LIN {X 4.349,Y -47.961,Z -134.902,A -90.000,B 90.000,C 0.000} C_DIS
LIN {X 3.638,Y -47.921,Z -134.978,A -90.000,B 90.000,C 0.000} C_DIS
LIN {X 3.458,Y -47.911,Z -134.966,A -90.000,B 90.000,C 0.000} C_DIS
LIN {X 3.249,Y -47.899,Z -134.959,A -90.000,B 90.000,C 0.000} C_DIS
LIN {X 3.035,Y -47.886,Z -134.959,A -90.000,B 90.000,C 0.000} C_DIS
LIN {X 2.734,Y -47.862,Z -134.966,A -90.000,B 90.000,C 0.000} C_DIS
LIN {X 2.521,Y -47.844,Z -134.907,A -90.000,B 90.000,C 0.000} C_DIS
LIN {X 2.240,Y -47.821,Z -134.818,A -90.000,B 90.000,C 0.000} C_DIS
LIN {X 1.961,Y -47.797,Z -134.712,A -90.000,B 90.000,C 0.000} C_DIS
LIN {X 1.753,Y -47.779,Z -134.622,A -90.000,B 90.000,C 0.000} C_DIS
LIN {X 1.325,Y -47.740,Z -134.399,A -90.000,B 90.000,C 0.000} C_DIS
LIN {X 1.040,Y -47.714,Z -134.237,A -90.000,B 90.000,C 0.000} C_DIS
LIN {X 0.850,Y -47.696,Z -134.116,A -90.000,B 90.000,C 0.000} C_DIS
LIN {X 0.755,Y -47.686,Z -134.050,A -90.000,B 90.000,C 0.000} C_DIS
LIN {X 0.661,Y -47.677,Z -133.981,A -90.000,B 90.000,C 0.000} C_DIS
LIN {X 0.569,Y -47.666,Z -133.907,A -90.000,B 90.000,C 0.000} C_DIS
LIN {X 0.394,Y -47.651,Z -133.762,A -90.000,B 90.000,C 0.000} C_DIS
LIN {X 0.029,Y -47.630,Z -133.079,A -90.000,B 90.000,C 0.000} C_DIS
LIN {X -0.030,Y -47.623,Z -132.969,A -90.000,B 90.000,C 0.000} C_DIS
LIN {X -0.099,Y -47.611,Z -132.836,A -90.000,B 90.000,C 0.000} C_DIS
LIN {X -0.133,Y -47.605,Z -132.740,A -90.000,B 90.000,C 0.000} C_DIS
LIN {X 0.043,Y -47.607,Z -130.577,A -90.000,B 90.000,C 0.000} C_DIS
LIN {X 0.099,Y -47.612,Z -130.301,A -90.000,B 90.000,C 0.000} C_DIS
LIN {X 0.135,Y -47.611,Z -130.125,A -90.000,B 90.000,C 0.000} C_DIS
LIN {X 0.250,Y -47.612,Z -129.925,A -90.000,B 90.000,C 0.000} C_DIS
LIN {X 1.143,Y -47.614,Z -128.527,A -90.000,B 90.000,C 0.000} C_DIS
LIN {X 1.838,Y -47.607,Z -127.443,A -90.000,B 90.000,C 0.000} C_DIS
LIN {X 2.056,Y -47.610,Z -127.175,A -90.000,B 90.000,C 0.000} C_DIS
LIN {X 2.200,Y -47.615,Z -127.035,A -90.000,B 90.000,C 0.000} C_DIS
LIN {X 2.268,Y -47.616,Z -126.970,A -90.000,B 90.000,C 0.000} C_DIS
LIN {X 3.440,Y -47.612,Z -125.853,A -90.000,B 90.000,C 0.000} C_DIS
LIN {X 3.637,Y -47.607,Z -125.667,A -90.000,B 90.000,C 0.000} C_DIS
LIN {X 4.260,Y -47.595,Z -125.097,A -90.000,B 90.000,C 0.000} C_DIS
LIN {X 4.386,Y -47.595,Z -125.003,A -90.000,B 90.000,C 0.000} C_DIS
LIN {X 5.546,Y -47.602,Z -124.204,A -90.000,B 90.000,C 0.000} C_DIS
LIN {X 5.853,Y -47.602,Z -123.993,A -90.000,B 90.000,C 0.000} C_DIS
LIN {X 6.516,Y -47.588,Z -123.540,A -90.000,B 90.000,C 0.000} C_DIS
LIN {X 6.563,Y -47.588,Z -123.512,A -90.000,B 90.000,C 0.000} C_DIS
LIN {X 8.622,Y -47.571,Z -122.476,A -90.000,B 90.000,C 0.000} C_DIS
LIN {X 9.750,Y -47.547,Z -121.910,A -90.000,B 90.000,C 0.000} C_DIS
LIN {X 12.160,Y -47.550,Z -121.167,A -90.000,B 90.000,C 0.000} C_DIS
LIN {X 14.408,Y -47.502,Z -120.480,A -90.000,B 90.000,C 0.000} C_DIS
LIN {X 14.547,Y -47.502,Z -120.468,A -90.000,B 90.000,C 0.000} C_DIS
LIN {X 16.833,Y -47.499,Z -120.228,A -90.000,B 90.000,C 0.000} C_DIS
LIN {X 17.033,Y -47.496,Z -120.208,A -90.000,B 90.000,C 0.000} C_DIS
LIN {X 18.502,Y -47.463,Z -120.057,A -90.000,B 90.000,C 0.000} C_DIS
LIN {X 18.616,Y -47.461,Z -120.057,A -90.000,B 90.000,C 0.000} C_DIS
LIN {X 21.308,Y -47.456,Z -120.534,A -90.000,B 90.000,C 0.000} C_DIS
LIN {X 21.567,Y -47.448,Z -120.581,A -90.000,B 90.000,C 0.000} C_DIS
LIN {X 21.787,Y -47.441,Z -120.626,A -90.000,B 90.000,C 0.000} C_DIS
LIN {X 22.175,Y -47.441,Z -120.928,A -90.000,B 90.000,C 0.000} C_DIS
LIN {X 23.178,Y -47.428,Z -121.711,A -90.000,B 90.000,C 0.000} C_DIS
LIN {X 23.442,Y -47.428,Z -122.009,A -90.000,B 90.000,C 0.000} C_DIS
LIN {X 23.523,Y -47.442,Z -122.462,A -90.000,B 90.000,C 0.000} C_DIS
LIN {X 23.482,Y -47.463,Z -122.835,A -90.000,B 90.000,C 0.000} C_DIS
LIN {X 23.458,Y -47.474,Z -123.058,A -90.000,B 90.000,C 0.000} C_DIS
LIN {X 23.449,Y -47.486,Z -123.390,A -90.000,B 90.000,C 0.000} C_DIS
LIN {X 23.488,Y -47.490,Z -123.844,A -90.000,B 90.000,C 0.000} C_DIS
LIN {X 23.560,Y -47.491,Z -124.679,A -90.000,B 90.000,C 0.000} C_DIS
LIN {X 23.397,Y -47.512,Z -125.426,A -90.000,B 90.000,C 0.000} C_DIS
LIN {X 23.214,Y -47.513,Z -126.253,A -90.000,B 90.000,C 0.000} C_DIS
LIN {X 23.157,Y -47.516,Z -126.512,A -90.000,B 90.000,C 0.000} C_DIS
LIN {X 22.471,Y -47.582,Z -127.926,A -90.000,B 90.000,C 0.000} C_DIS
LIN {X 22.078,Y -47.598,Z -128.731,A -90.000,B 90.000,C 0.000} C_DIS
LIN {X 21.868,Y -47.607,Z -129.140,A -90.000,B 90.000,C 0.000} C_DIS
LIN {X 21.688,Y -47.619,Z -129.394,A -90.000,B 90.000,C 0.000} C_DIS
LIN {X 20.899,Y -47.663,Z -130.579,A -90.000,B 90.000,C 0.000} C_DIS
LIN {X 20.391,Y -47.672,Z -131.337,A -90.000,B 90.000,C 0.000} C_DIS
LIN {X 19.805,Y -47.696,Z -132.023,A -90.000,B 90.000,C 0.000} C_DIS
LIN {X 19.346,Y -47.720,Z -132.478,A -90.000,B 90.000,C 0.000} C_DIS
LIN {X 18.457,Y -47.730,Z -133.348,A -90.000,B 90.000,C 0.000} C_DIS
LIN {X 18.205,Y -47.729,Z -133.593,A -90.000,B 90.000,C 0.000} C_DIS
LIN {X 17.590,Y -47.732,Z -134.145,A -90.000,B 90.000,C 0.000} C_DIS
LIN {X 17.544,Y -47.732,Z -134.183,A -90.000,B 90.000,C 0.000} C_DIS
LIN {X 17.409,Y -47.738,Z -134.263,A -90.000,B 90.000,C 0.000} C_DIS
LIN {X 17.214,Y -47.749,Z -134.364,A -90.000,B 90.000,C 0.000} C_DIS
LIN {X 16.932,Y -47.764,Z -134.516,A -90.000,B 90.000,C 0.000} C_DIS
LIN {X 16.164,Y -47.806,Z -134.922,A -90.000,B 90.000,C 0.000} C_DIS
LIN {X 15.908,Y -47.817,Z -135.056,A -90.000,B 90.000,C 0.000} C_DIS
LIN {X 15.083,Y -47.818,Z -135.479,A -90.000,B 90.000,C 0.000} C_DIS
LIN {X 14.959,Y -47.815,Z -135.542,A -90.000,B 90.000,C 0.000} C_DIS
LIN {X 13.972,Y -47.784,Z -136.033,A -90.000,B 90.000,C 0.000} C_DIS
LIN {X 13.915,Y -47.784,Z -136.053,A -90.000,B 90.000,C 0.000} C_DIS
LIN {X 13.450,Y -47.784,Z -136.207,A -90.000,B 90.000,C 0.000} C_DIS
LIN {X 13.362,Y -47.784,Z -136.234,A -90.000,B 90.000,C 0.000} C_DIS
LIN {X 13.341,Y -47.785,Z -136.240,A -90.000,B 90.000,C 0.000} C_DIS
LIN {X 12.439,Y -47.811,Z -136.397,A -90.000,B 90.000,C 0.000} C_DIS
LIN {X 10.398,Y -47.880,Z -136.688,A -90.000,B 90.000,C 0.000} C_DIS
LIN {X 10.207,Y -47.881,Z -136.713,A -90.000,B 90.000,C 0.000} C_DIS
LIN {X 9.590,Y -47.863,Z -136.790,A -90.000,B 90.000,C 0.000} C_DIS
LIN {X 8.229,Y -47.857,Z -136.774,A -90.000,B 90.000,C 0.000} C_DIS
LIN {X 7.049,Y -47.839,Z -136.755,A -90.000,B 90.000,C 0.000} C_DIS
LIN {X 6.522,Y -47.832,Z -136.740,A -90.000,B 90.000,C 0.000} C_DIS
LIN {X 6.298,Y -47.824,Z -136.732,A -90.000,B 90.000,C 0.000} C_DIS
LIN {X 6.019,Y -47.803,Z -136.719,A -90.000,B 90.000,C 0.000} C_DIS
LIN {X 5.735,Y -47.783,Z -136.693,A -90.000,B 90.000,C 0.000} C_DIS
LIN {X 5.512,Y -47.783,Z -136.604,A -90.000,B 90.000,C 0.000} C_DIS
LIN {X 5.374,Y -47.782,Z -136.555,A -90.000,B 90.000,C 0.000} C_DIS
LIN {X 3.264,Y -47.744,Z -135.889,A -90.000,B 90.000,C 0.000} C_DIS
LIN {X 3.000,Y -47.743,Z -135.807,A -90.000,B 90.000,C 0.000} C_DIS
LIN {X 2.785,Y -47.739,Z -135.739,A -90.000,B 90.000,C 0.000} C_DIS
LIN {X 2.660,Y -47.732,Z -135.698,A -90.000,B 90.000,C 0.000} C_DIS
LIN {X 2.579,Y -47.735,Z -135.627,A -90.000,B 90.000,C 0.000} C_DIS
LIN {X 2.188,Y -47.735,Z -135.280,A -90.000,B 90.000,C 0.000} C_DIS
LIN {X 1.658,Y -47.726,Z -134.806,A -90.000,B 90.000,C 0.000} C_DIS
LIN {X 1.300,Y -47.717,Z -134.512,A -90.000,B 90.000,C 0.000} C_DIS
LIN {X 1.078,Y -47.706,Z -134.329,A -90.000,B 90.000,C 0.000} C_DIS
LIN {X 0.956,Y -47.697,Z -134.228,A -90.000,B 90.000,C 0.000} C_DIS
LIN {X 0.569,Y -47.666,Z -133.907,A -90.000,B 90.000,C 0.000} C_DIS
LIN {X 0.393,Y -47.657,Z -133.765,A -90.000,B 90.000,C 0.000} C_DIS
LIN {X 0.270,Y -47.647,Z -133.556,A -90.000,B 90.000,C 0.000} C_DIS
LIN {X 0.189,Y -47.641,Z -133.425,A -90.000,B 90.000,C 0.000} C_DIS
LIN {X 0.021,Y -47.629,Z -133.169,A -90.000,B 90.000,C 0.000} C_DIS
LIN {X -0.161,Y -47.616,Z -132.904,A -90.000,B 90.000,C 0.000} C_DIS
LIN {X -0.203,Y -47.612,Z -132.822,A -90.000,B 90.000,C 0.000} C_DIS
LIN {X -0.214,Y -47.605,Z -132.651,A -90.000,B 90.000,C 0.000} C_DIS
LIN {X -0.228,Y -47.600,Z -132.517,A -90.000,B 90.000,C 0.000} C_DIS
LIN {X -0.255,Y -47.592,Z -132.319,A -90.000,B 90.000,C 0.000} C_DIS
LIN {X -0.278,Y -47.586,Z -132.189,A -90.000,B 90.000,C 0.000} C_DIS
LIN {X -0.318,Y -47.579,Z -131.998,A -90.000,B 90.000,C 0.000} C_DIS
LIN {X -0.349,Y -47.573,Z -131.872,A -90.000,B 90.000,C 0.000} C_DIS
LIN {X -0.420,Y -47.563,Z -131.624,A -90.000,B 90.000,C 0.000} C_DIS
LIN {X -0.560,Y -47.540,Z -131.077,A -90.000,B 90.000,C 0.000} C_DIS
LIN {X -0.623,Y -47.526,Z -130.741,A -90.000,B 90.000,C 0.000} C_DIS
LIN {X -0.614,Y -47.515,Z -130.467,A -90.000,B 90.000,C 0.000} C_DIS
LIN {X -0.615,Y -47.511,Z -130.363,A -90.000,B 90.000,C 0.000} C_DIS
LIN {X -0.627,Y -47.502,Z -130.152,A -90.000,B 90.000,C 0.000} C_DIS
LIN {X -0.654,Y -47.493,Z -129.936,A -90.000,B 90.000,C 0.000} C_DIS
LIN {X -0.672,Y -47.488,Z -129.827,A -90.000,B 90.000,C 0.000} C_DIS
LIN {X -0.704,Y -47.480,Z -129.660,A -90.000,B 90.000,C 0.000} C_DIS
LIN {X -0.743,Y -47.466,Z -129.380,A -90.000,B 90.000,C 0.000} C_DIS
LIN {X -0.791,Y -47.452,Z -129.092,A -90.000,B 90.000,C 0.000} C_DIS
LIN {X -0.801,Y -47.447,Z -128.991,A -90.000,B 90.000,C 0.000} C_DIS
LIN {X -0.783,Y -47.438,Z -128.816,A -90.000,B 90.000,C 0.000} C_DIS
LIN {X -0.768,Y -47.433,Z -128.708,A -90.000,B 90.000,C 0.000} C_DIS
LIN {X -0.752,Y -47.427,Z -128.600,A -90.000,B 90.000,C 0.000} C_DIS
LIN {X -0.728,Y -47.422,Z -128.495,A -90.000,B 90.000,C 0.000} C_DIS
LIN {X -0.671,Y -47.411,Z -128.283,A -90.000,B 90.000,C 0.000} C_DIS
LIN {X -0.604,Y -47.400,Z -128.068,A -90.000,B 90.000,C 0.000} C_DIS
LIN {X -0.529,Y -47.389,Z -127.846,A -90.000,B 90.000,C 0.000} C_DIS
LIN {X -0.445,Y -47.377,Z -127.616,A -90.000,B 90.000,C 0.000} C_DIS
LIN {X -0.351,Y -47.364,Z -127.380,A -90.000,B 90.000,C 0.000} C_DIS
LIN {X -0.299,Y -47.358,Z -127.259,A -90.000,B 90.000,C 0.000} C_DIS
LIN {X -0.184,Y -47.345,Z -127.012,A -90.000,B 90.000,C 0.000} C_DIS
LIN {X -0.053,Y -47.331,Z -126.758,A -90.000,B 90.000,C 0.000} C_DIS
LIN {X 0.020,Y -47.323,Z -126.629,A -90.000,B 90.000,C 0.000} C_DIS
LIN {X 0.179,Y -47.308,Z -126.366,A -90.000,B 90.000,C 0.000} C_DIS
LIN {X 0.233,Y -47.308,Z -126.282,A -90.000,B 90.000,C 0.000} C_DIS
LIN {X 0.581,Y -47.308,Z -125.855,A -90.000,B 90.000,C 0.000} C_DIS
LIN {X 0.688,Y -47.308,Z -125.746,A -90.000,B 90.000,C 0.000} C_DIS
LIN {X 2.304,Y -47.308,Z -124.205,A -90.000,B 90.000,C 0.000} C_DIS
LIN {X 2.998,Y -47.308,Z -123.569,A -90.000,B 90.000,C 0.000} C_DIS
LIN {X 3.235,Y -47.308,Z -123.392,A -90.000,B 90.000,C 0.000} C_DIS
LIN {X 5.471,Y -47.308,Z -121.855,A -90.000,B 90.000,C 0.000} C_DIS
LIN {X 5.627,Y -47.308,Z -121.766,A -90.000,B 90.000,C 0.000} C_DIS
LIN {X 9.005,Y -47.308,Z -120.061,A -90.000,B 90.000,C 0.000} C_DIS
LIN {X 13.904,Y -47.308,Z -118.552,A -90.000,B 90.000,C 0.000} C_DIS
LIN {X 14.072,Y -47.308,Z -118.512,A -90.000,B 90.000,C 0.000} C_DIS
LIN {X 14.371,Y -47.308,Z -118.485,A -90.000,B 90.000,C 0.000} C_DIS
LIN {X 18.398,Y -47.308,Z -118.063,A -90.000,B 90.000,C 0.000} C_DIS
LIN {X 18.792,Y -47.308,Z -118.063,A -90.000,B 90.000,C 0.000} C_DIS
LIN {X 21.939,Y -47.308,Z -118.620,A -90.000,B 90.000,C 0.000} C_DIS
LIN {X 22.643,Y -47.308,Z -118.763,A -90.000,B 90.000,C 0.000} C_DIS
LIN {X 24.510,Y -47.308,Z -120.218,A -90.000,B 90.000,C 0.000} C_DIS
LIN {X 24.576,Y -47.308,Z -120.277,A -90.000,B 90.000,C 0.000} C_DIS
LIN {X 25.298,Y -47.308,Z -121.096,A -90.000,B 90.000,C 0.000} C_DIS
LIN {X 25.323,Y -47.308,Z -121.181,A -90.000,B 90.000,C 0.000} C_DIS
LIN {X 25.538,Y -47.308,Z -122.399,A -90.000,B 90.000,C 0.000} C_DIS
LIN {X 25.438,Y -47.308,Z -123.282,A -90.000,B 90.000,C 0.000} C_DIS
LIN {X 25.566,Y -47.308,Z -124.764,A -90.000,B 90.000,C 0.000} C_DIS
LIN {X 25.558,Y -47.308,Z -124.867,A -90.000,B 90.000,C 0.000} C_DIS
LIN {X 25.073,Y -47.308,Z -127.058,A -90.000,B 90.000,C 0.000} C_DIS
LIN {X 25.021,Y -47.308,Z -127.227,A -90.000,B 90.000,C 0.000} C_DIS
LIN {X 25.004,Y -47.308,Z -127.267,A -90.000,B 90.000,C 0.000} C_DIS
LIN {X 24.995,Y -47.308,Z -127.282,A -90.000,B 90.000,C 0.000} C_DIS
LIN {X 23.838,Y -47.308,Z -129.636,A -90.000,B 90.000,C 0.000} C_DIS
LIN {X 23.694,Y -47.308,Z -129.917,A -90.000,B 90.000,C 0.000} C_DIS
LIN {X 23.558,Y -47.308,Z -130.176,A -90.000,B 90.000,C 0.000} C_DIS
LIN {X 23.296,Y -47.308,Z -130.542,A -90.000,B 90.000,C 0.000} C_DIS
LIN {X 21.965,Y -47.308,Z -132.519,A -90.000,B 90.000,C 0.000} C_DIS
LIN {X 21.855,Y -47.308,Z -132.651,A -90.000,B 90.000,C 0.000} C_DIS
LIN {X 21.236,Y -47.308,Z -133.369,A -90.000,B 90.000,C 0.000} C_DIS
LIN {X 19.541,Y -47.308,Z -135.022,A -90.000,B 90.000,C 0.000} C_DIS
LIN {X 18.869,Y -47.308,Z -135.624,A -90.000,B 90.000,C 0.000} C_DIS
LIN {X 18.653,Y -47.308,Z -135.802,A -90.000,B 90.000,C 0.000} C_DIS
LIN {X 18.421,Y -47.308,Z -135.934,A -90.000,B 90.000,C 0.000} C_DIS
LIN {X 17.821,Y -47.308,Z -136.249,A -90.000,B 90.000,C 0.000} C_DIS
LIN {X 15.640,Y -47.308,Z -137.367,A -90.000,B 90.000,C 0.000} C_DIS
LIN {X 14.735,Y -47.308,Z -137.824,A -90.000,B 90.000,C 0.000} C_DIS
LIN {X 14.524,Y -47.308,Z -137.898,A -90.000,B 90.000,C 0.000} C_DIS
LIN {X 13.952,Y -47.308,Z -138.087,A -90.000,B 90.000,C 0.000} C_DIS
LIN {X 13.796,Y -47.308,Z -138.129,A -90.000,B 90.000,C 0.000} C_DIS
LIN {X 13.757,Y -47.308,Z -138.140,A -90.000,B 90.000,C 0.000} C_DIS
LIN {X 12.690,Y -47.308,Z -138.317,A -90.000,B 90.000,C 0.000} C_DIS
LIN {X 9.707,Y -47.308,Z -138.712,A -90.000,B 90.000,C 0.000} C_DIS
LIN {X 7.282,Y -47.308,Z -138.687,A -90.000,B 90.000,C 0.000} C_DIS
LIN {X 7.000,Y -47.308,Z -138.683,A -90.000,B 90.000,C 0.000} C_DIS
LIN {X 5.923,Y -47.308,Z -138.655,A -90.000,B 90.000,C 0.000} C_DIS
LIN {X 5.452,Y -47.308,Z -138.620,A -90.000,B 90.000,C 0.000} C_DIS
LIN {X 5.219,Y -47.308,Z -138.578,A -90.000,B 90.000,C 0.000} C_DIS
LIN {X 4.796,Y -47.308,Z -138.410,A -90.000,B 90.000,C 0.000} C_DIS
LIN {X 1.927,Y -47.308,Z -137.517,A -90.000,B 90.000,C 0.000} C_DIS
LIN {X 1.708,Y -47.308,Z -137.427,A -90.000,B 90.000,C 0.000} C_DIS
LIN {X 1.512,Y -47.308,Z -137.293,A -90.000,B 90.000,C 0.000} C_DIS
LIN {X 0.365,Y -47.308,Z -136.273,A -90.000,B 90.000,C 0.000} C_DIS
LIN {X -1.002,Y -47.308,Z -135.167,A -90.000,B 90.000,C 0.000} C_DIS
LIN {X -1.165,Y -47.308,Z -134.995,A -90.000,B 90.000,C 0.000} C_DIS
LIN {X -1.289,Y -47.308,Z -134.793,A -90.000,B 90.000,C 0.000} C_DIS
LIN {X -1.910,Y -47.308,Z -133.644,A -90.000,B 90.000,C 0.000} C_DIS
LIN {X -2.118,Y -47.308,Z -133.061,A -90.000,B 90.000,C 0.000} C_DIS
LIN {X -2.129,Y -47.308,Z -132.882,A -90.000,B 90.000,C 0.000} C_DIS
LIN {X -1.918,Y -47.308,Z -130.298,A -90.000,B 90.000,C 0.000} C_DIS
LIN {X -1.761,Y -47.308,Z -129.531,A -90.000,B 90.000,C 0.000} C_DIS
LIN {X -1.718,Y -47.308,Z -129.388,A -90.000,B 90.000,C 0.000} C_DIS
LIN {X -1.614,Y -47.308,Z -129.199,A -90.000,B 90.000,C 0.000} C_DIS
LIN {X -1.441,Y -47.308,Z -128.899,A -90.000,B 90.000,C 0.000} C_DIS
LIN {X 0.179,Y -47.308,Z -126.366,A -90.000,B 90.000,C 0.000} C_DIS
LIN {X 0.233,Y -47.313,Z -126.281,A -90.000,B 90.000,C 0.000} C_DIS
LIN {X 0.390,Y -47.313,Z -126.081,A -90.000,B 90.000,C 0.000} C_DIS
LIN {X 0.561,Y -47.310,Z -125.850,A -90.000,B 90.000,C 0.000} C_DIS
LIN {X 0.836,Y -47.303,Z -125.538,A -90.000,B 90.000,C 0.000} C_DIS
LIN {X 1.062,Y -47.297,Z -125.273,A -90.000,B 90.000,C 0.000} C_DIS
LIN {X 1.280,Y -47.290,Z -125.003,A -90.000,B 90.000,C 0.000} C_DIS
LIN {X 1.492,Y -47.281,Z -124.728,A -90.000,B 90.000,C 0.000} C_DIS
LIN {X 1.697,Y -47.271,Z -124.450,A -90.000,B 90.000,C 0.000} C_DIS
LIN {X 1.897,Y -47.262,Z -124.167,A -90.000,B 90.000,C 0.000} C_DIS
LIN {X 2.191,Y -47.248,Z -123.742,A -90.000,B 90.000,C 0.000} C_DIS
LIN {X 2.514,Y -47.232,Z -123.260,A -90.000,B 90.000,C 0.000} C_DIS
LIN {X 2.679,Y -47.224,Z -123.041,A -90.000,B 90.000,C 0.000} C_DIS
LIN {X 2.885,Y -47.215,Z -122.777,A -90.000,B 90.000,C 0.000} C_DIS
LIN {X 3.512,Y -47.187,Z -122.001,A -90.000,B 90.000,C 0.000} C_DIS
LIN {X 3.933,Y -47.169,Z -121.488,A -90.000,B 90.000,C 0.000} C_DIS
LIN {X 4.251,Y -47.156,Z -121.106,A -90.000,B 90.000,C 0.000} C_DIS
LIN {X 4.360,Y -47.151,Z -120.981,A -90.000,B 90.000,C 0.000} C_DIS
LIN {X 4.778,Y -47.134,Z -120.527,A -90.000,B 90.000,C 0.000} C_DIS
LIN {X 4.894,Y -47.129,Z -120.410,A -90.000,B 90.000,C 0.000} C_DIS
LIN {X 5.014,Y -47.125,Z -120.299,A -90.000,B 90.000,C 0.000} C_DIS
LIN {X 5.293,Y -47.115,Z -120.063,A -90.000,B 90.000,C 0.000} C_DIS
LIN {X 5.678,Y -47.101,Z -119.758,A -90.000,B 90.000,C 0.000} C_DIS
LIN {X 5.943,Y -47.092,Z -119.561,A -90.000,B 90.000,C 0.000} C_DIS
LIN {X 6.078,Y -47.088,Z -119.465,A -90.000,B 90.000,C 0.000} C_DIS
LIN {X 6.353,Y -47.079,Z -119.275,A -90.000,B 90.000,C 0.000} C_DIS
LIN {X 6.494,Y -47.074,Z -119.183,A -90.000,B 90.000,C 0.000} C_DIS
LIN {X 6.782,Y -47.065,Z -119.002,A -90.000,B 90.000,C 0.000} C_DIS
LIN {X 7.079,Y -47.055,Z -118.828,A -90.000,B 90.000,C 0.000} C_DIS
LIN {X 7.231,Y -47.050,Z -118.743,A -90.000,B 90.000,C 0.000} C_DIS
LIN {X 7.542,Y -47.041,Z -118.579,A -90.000,B 90.000,C 0.000} C_DIS
LIN {X 8.112,Y -47.042,Z -118.292,A -90.000,B 90.000,C 0.000} C_DIS
LIN {X 8.422,Y -47.046,Z -118.166,A -90.000,B 90.000,C 0.000} C_DIS
LIN {X 10.316,Y -47.086,Z -117.578,A -90.000,B 90.000,C 0.000} C_DIS
LIN {X 10.927,Y -47.095,Z -117.389,A -90.000,B 90.000,C 0.000} C_DIS
LIN {X 13.319,Y -47.092,Z -116.652,A -90.000,B 90.000,C 0.000} C_DIS
LIN {X 13.423,Y -47.092,Z -116.623,A -90.000,B 90.000,C 0.000} C_DIS
LIN {X 13.602,Y -47.094,Z -116.579,A -90.000,B 90.000,C 0.000} C_DIS
LIN {X 13.823,Y -47.096,Z -116.538,A -90.000,B 90.000,C 0.000} C_DIS
LIN {X 14.179,Y -47.104,Z -116.505,A -90.000,B 90.000,C 0.000} C_DIS
LIN {X 15.609,Y -47.133,Z -116.352,A -90.000,B 90.000,C 0.000} C_DIS
LIN {X 17.666,Y -47.130,Z -116.136,A -90.000,B 90.000,C 0.000} C_DIS
LIN {X 18.223,Y -47.133,Z -116.078,A -90.000,B 90.000,C 0.000} C_DIS
LIN {X 18.399,Y -47.134,Z -116.070,A -90.000,B 90.000,C 0.000} C_DIS
LIN {X 18.793,Y -47.139,Z -116.070,A -90.000,B 90.000,C 0.000} C_DIS
LIN {X 19.140,Y -47.146,Z -116.100,A -90.000,B 90.000,C 0.000} C_DIS
LIN {X 20.083,Y -47.169,Z -116.265,A -90.000,B 90.000,C 0.000} C_DIS
LIN {X 22.335,Y -47.177,Z -116.664,A -90.000,B 90.000,C 0.000} C_DIS
LIN {X 23.040,Y -47.180,Z -116.807,A -90.000,B 90.000,C 0.000} C_DIS
LIN {X 23.322,Y -47.183,Z -116.886,A -90.000,B 90.000,C 0.000} C_DIS
LIN {X 23.626,Y -47.189,Z -117.025,A -90.000,B 90.000,C 0.000} C_DIS
LIN {X 23.766,Y -47.193,Z -117.112,A -90.000,B 90.000,C 0.000} C_DIS
LIN {X 23.856,Y -47.195,Z -117.177,A -90.000,B 90.000,C 0.000} C_DIS
LIN {X 24.910,Y -47.194,Z -117.998,A -90.000,B 90.000,C 0.000} C_DIS
LIN {X 25.752,Y -47.189,Z -118.655,A -90.000,B 90.000,C 0.000} C_DIS
LIN {X 25.850,Y -47.188,Z -118.738,A -90.000,B 90.000,C 0.000} C_DIS
LIN {X 25.908,Y -47.188,Z -118.790,A -90.000,B 90.000,C 0.000} C_DIS
LIN {X 26.003,Y -47.188,Z -118.881,A -90.000,B 90.000,C 0.000} C_DIS
LIN {X 26.074,Y -47.189,Z -118.957,A -90.000,B 90.000,C 0.000} C_DIS
LIN {X 26.562,Y -47.192,Z -119.510,A -90.000,B 90.000,C 0.000} C_DIS
LIN {X 26.795,Y -47.179,Z -119.776,A -90.000,B 90.000,C 0.000} C_DIS
LIN {X 26.950,Y -47.168,Z -119.977,A -90.000,B 90.000,C 0.000} C_DIS
LIN {X 27.026,Y -47.162,Z -120.098,A -90.000,B 90.000,C 0.000} C_DIS
LIN {X 27.105,Y -47.158,Z -120.252,A -90.000,B 90.000,C 0.000} C_DIS
LIN {X 27.129,Y -47.157,Z -120.305,A -90.000,B 90.000,C 0.000} C_DIS
LIN {X 27.215,Y -47.154,Z -120.545,A -90.000,B 90.000,C 0.000} C_DIS
LIN {X 27.239,Y -47.153,Z -120.630,A -90.000,B 90.000,C 0.000} C_DIS
LIN {X 27.286,Y -47.152,Z -120.834,A -90.000,B 90.000,C 0.000} C_DIS
LIN {X 27.478,Y -47.151,Z -121.920,A -90.000,B 90.000,C 0.000} C_DIS
LIN {X 27.508,Y -47.147,Z -122.093,A -90.000,B 90.000,C 0.000} C_DIS
LIN {X 27.524,Y -47.144,Z -122.225,A -90.000,B 90.000,C 0.000} C_DIS
LIN {X 27.531,Y -47.142,Z -122.369,A -90.000,B 90.000,C 0.000} C_DIS
LIN {X 27.525,Y -47.141,Z -122.555,A -90.000,B 90.000,C 0.000} C_DIS
LIN {X 27.468,Y -47.141,Z -123.074,A -90.000,B 90.000,C 0.000} C_DIS
LIN {X 27.441,Y -47.141,Z -123.309,A -90.000,B 90.000,C 0.000} C_DIS
LIN {X 27.527,Y -47.123,Z -124.323,A -90.000,B 90.000,C 0.000} C_DIS
LIN {X 27.539,Y -47.114,Z -124.471,A -90.000,B 90.000,C 0.000} C_DIS
LIN {X 27.554,Y -47.099,Z -124.680,A -90.000,B 90.000,C 0.000} C_DIS
LIN {X 27.547,Y -47.084,Z -124.923,A -90.000,B 90.000,C 0.000} C_DIS
LIN {X 27.539,Y -47.079,Z -125.025,A -90.000,B 90.000,C 0.000} C_DIS
LIN {X 27.497,Y -47.068,Z -125.296,A -90.000,B 90.000,C 0.000} C_DIS
LIN {X 27.188,Y -47.028,Z -126.666,A -90.000,B 90.000,C 0.000} C_DIS
LIN {X 26.985,Y -46.969,Z -127.539,A -90.000,B 90.000,C 0.000} C_DIS
LIN {X 26.902,Y -46.953,Z -127.807,A -90.000,B 90.000,C 0.000} C_DIS
LIN {X 26.817,Y -46.943,Z -128.029,A -90.000,B 90.000,C 0.000} C_DIS
LIN {X 26.762,Y -46.939,Z -128.147,A -90.000,B 90.000,C 0.000} C_DIS
LIN {X 26.726,Y -46.939,Z -128.215,A -90.000,B 90.000,C 0.000} C_DIS
LIN {X 26.204,Y -46.937,Z -129.278,A -90.000,B 90.000,C 0.000} C_DIS
LIN {X 26.139,Y -46.936,Z -129.410,A -90.000,B 90.000,C 0.000} C_DIS
LIN {X 25.577,Y -46.892,Z -130.532,A -90.000,B 90.000,C 0.000} C_DIS
LIN {X 25.287,Y -46.873,Z -131.083,A -90.000,B 90.000,C 0.000} C_DIS
LIN {X 25.269,Y -46.872,Z -131.114,A -90.000,B 90.000,C 0.000} C_DIS
LIN {X 25.173,Y -46.870,Z -131.270,A -90.000,B 90.000,C 0.000} C_DIS
LIN {X 24.900,Y -46.871,Z -131.655,A -90.000,B 90.000,C 0.000} C_DIS
LIN {X 24.020,Y -46.825,Z -132.942,A -90.000,B 90.000,C 0.000} C_DIS
LIN {X 23.560,Y -46.796,Z -133.612,A -90.000,B 90.000,C 0.000} C_DIS
LIN {X 23.449,Y -46.793,Z -133.758,A -90.000,B 90.000,C 0.000} C_DIS
LIN {X 23.317,Y -46.791,Z -133.914,A -90.000,B 90.000,C 0.000} C_DIS
LIN {X 23.115,Y -46.790,Z -134.148,A -90.000,B 90.000,C 0.000} C_DIS
LIN {X 22.837,Y -46.776,Z -134.463,A -90.000,B 90.000,C 0.000} C_DIS
LIN {X 22.693,Y -46.765,Z -134.626,A -90.000,B 90.000,C 0.000} C_DIS
LIN {X 22.566,Y -46.758,Z -134.757,A -90.000,B 90.000,C 0.000} C_DIS
LIN {X 20.843,Y -46.702,Z -136.414,A -90.000,B 90.000,C 0.000} C_DIS
LIN {X 20.684,Y -46.691,Z -136.552,A -90.000,B 90.000,C 0.000} C_DIS
LIN {X 20.126,Y -46.641,Z -137.029,A -90.000,B 90.000,C 0.000} C_DIS
LIN {X 19.851,Y -46.621,Z -137.249,A -90.000,B 90.000,C 0.000} C_DIS
LIN {X 19.642,Y -46.613,Z -137.395,A -90.000,B 90.000,C 0.000} C_DIS
LIN {X 19.293,Y -46.616,Z -137.595,A -90.000,B 90.000,C 0.000} C_DIS
LIN {X 18.679,Y -46.629,Z -137.923,A -90.000,B 90.000,C 0.000} C_DIS
LIN {X 17.979,Y -46.647,Z -138.289,A -90.000,B 90.000,C 0.000} C_DIS
LIN {X 17.207,Y -46.637,Z -138.681,A -90.000,B 90.000,C 0.000} C_DIS
LIN {X 16.900,Y -46.623,Z -138.832,A -90.000,B 90.000,C 0.000} C_DIS
LIN {X 16.480,Y -46.594,Z -139.036,A -90.000,B 90.000,C 0.000} C_DIS
LIN {X 15.565,Y -46.534,Z -139.470,A -90.000,B 90.000,C 0.000} C_DIS
LIN {X 15.345,Y -46.526,Z -139.560,A -90.000,B 90.000,C 0.000} C_DIS
LIN {X 15.099,Y -46.524,Z -139.646,A -90.000,B 90.000,C 0.000} C_DIS
LIN {X 14.529,Y -46.523,Z -139.834,A -90.000,B 90.000,C 0.000} C_DIS
LIN {X 14.437,Y -46.524,Z -139.862,A -90.000,B 90.000,C 0.000} C_DIS
LIN {X 14.242,Y -46.528,Z -139.917,A -90.000,B 90.000,C 0.000} C_DIS
LIN {X 14.058,Y -46.535,Z -139.960,A -90.000,B 90.000,C 0.000} C_DIS
LIN {X 13.283,Y -46.575,Z -140.105,A -90.000,B 90.000,C 0.000} C_DIS
LIN {X 13.106,Y -46.582,Z -140.137,A -90.000,B 90.000,C 0.000} C_DIS
LIN {X 12.935,Y -46.584,Z -140.165,A -90.000,B 90.000,C 0.000} C_DIS
LIN {X 11.458,Y -46.596,Z -140.366,A -90.000,B 90.000,C 0.000} C_DIS
LIN {X 9.952,Y -46.584,Z -140.560,A -90.000,B 90.000,C 0.000} C_DIS
LIN {X 9.686,Y -46.590,Z -140.579,A -90.000,B 90.000,C 0.000} C_DIS
LIN {X 9.181,Y -46.616,Z -140.584,A -90.000,B 90.000,C 0.000} C_DIS
LIN {X 8.870,Y -46.625,Z -140.584,A -90.000,B 90.000,C 0.000} C_DIS
LIN {X 8.155,Y -46.630,Z -140.578,A -90.000,B 90.000,C 0.000} C_DIS
LIN {X 6.969,Y -46.616,Z -140.559,A -90.000,B 90.000,C 0.000} C_DIS
LIN {X 5.809,Y -46.609,Z -140.526,A -90.000,B 90.000,C 0.000} C_DIS
LIN {X 5.311,Y -46.615,Z -140.491,A -90.000,B 90.000,C 0.000} C_DIS
LIN {X 5.107,Y -46.622,Z -140.466,A -90.000,B 90.000,C 0.000} C_DIS
LIN {X 4.884,Y -46.630,Z -140.429,A -90.000,B 90.000,C 0.000} C_DIS
LIN {X 4.813,Y -46.633,Z -140.416,A -90.000,B 90.000,C 0.000} C_DIS
LIN {X 4.689,Y -46.640,Z -140.387,A -90.000,B 90.000,C 0.000} C_DIS
LIN {X 4.553,Y -46.647,Z -140.344,A -90.000,B 90.000,C 0.000} C_DIS
LIN {X 4.430,Y -46.655,Z -140.298,A -90.000,B 90.000,C 0.000} C_DIS
LIN {X 4.165,Y -46.667,Z -140.198,A -90.000,B 90.000,C 0.000} C_DIS
LIN {X 2.337,Y -46.696,Z -139.639,A -90.000,B 90.000,C 0.000} C_DIS
LIN {X 1.358,Y -46.731,Z -139.346,A -90.000,B 90.000,C 0.000} C_DIS
LIN {X 1.239,Y -46.737,Z -139.306,A -90.000,B 90.000,C 0.000} C_DIS
LIN {X 1.036,Y -46.750,Z -139.228,A -90.000,B 90.000,C 0.000} C_DIS
LIN {X 0.977,Y -46.751,Z -139.204,A -90.000,B 90.000,C 0.000} C_DIS
LIN {X 0.856,Y -46.753,Z -139.150,A -90.000,B 90.000,C 0.000} C_DIS
LIN {X 0.782,Y -46.756,Z -139.112,A -90.000,B 90.000,C 0.000} C_DIS
LIN {X 0.747,Y -46.756,Z -139.092,A -90.000,B 90.000,C 0.000} C_DIS
LIN {X 0.620,Y -46.759,Z -139.013,A -90.000,B 90.000,C 0.000} C_DIS
LIN {X 0.424,Y -46.766,Z -138.881,A -90.000,B 90.000,C 0.000} C_DIS
LIN {X 0.288,Y -46.773,Z -138.782,A -90.000,B 90.000,C 0.000} C_DIS
LIN {X 0.204,Y -46.781,Z -138.712,A -90.000,B 90.000,C 0.000} C_DIS
LIN {X -0.726,Y -46.867,Z -137.913,A -90.000,B 90.000,C 0.000} C_DIS
LIN {X -0.899,Y -46.880,Z -137.763,A -90.000,B 90.000,C 0.000} C_DIS
LIN {X -1.681,Y -46.919,Z -137.141,A -90.000,B 90.000,C 0.000} C_DIS
LIN {X -1.816,Y -46.922,Z -137.033,A -90.000,B 90.000,C 0.000} C_DIS
LIN {X -2.122,Y -46.922,Z -136.785,A -90.000,B 90.000,C 0.000} C_DIS
LIN {X -2.299,Y -46.916,Z -136.638,A -90.000,B 90.000,C 0.000} C_DIS
LIN {X -2.353,Y -46.912,Z -136.588,A -90.000,B 90.000,C 0.000} C_DIS
LIN {X -2.448,Y -46.905,Z -136.490,A -90.000,B 90.000,C 0.000} C_DIS
LIN {X -2.585,Y -46.895,Z -136.342,A -90.000,B 90.000,C 0.000} C_DIS
LIN {X -2.712,Y -46.887,Z -136.191,A -90.000,B 90.000,C 0.000} C_DIS
LIN {X -2.833,Y -46.884,Z -136.014,A -90.000,B 90.000,C 0.000} C_DIS
LIN {X -2.956,Y -46.882,Z -135.811,A -90.000,B 90.000,C 0.000} C_DIS
LIN {X -3.007,Y -46.882,Z -135.722,A -90.000,B 90.000,C 0.000} C_DIS
LIN {X -3.586,Y -46.885,Z -134.655,A -90.000,B 90.000,C 0.000} C_DIS
LIN {X -3.661,Y -46.886,Z -134.514,A -90.000,B 90.000,C 0.000} C_DIS
LIN {X -3.722,Y -46.889,Z -134.378,A -90.000,B 90.000,C 0.000} C_DIS
LIN {X -3.752,Y -46.891,Z -134.301,A -90.000,B 90.000,C 0.000} C_DIS
LIN {X -3.964,Y -46.911,Z -133.720,A -90.000,B 90.000,C 0.000} C_DIS
LIN {X -4.058,Y -46.929,Z -133.368,A -90.000,B 90.000,C 0.000} C_DIS
LIN {X -4.070,Y -46.935,Z -133.288,A -90.000,B 90.000,C 0.000} C_DIS
LIN {X -4.080,Y -46.941,Z -133.178,A -90.000,B 90.000,C 0.000} C_DIS
LIN {X -4.093,Y -46.951,Z -132.991,A -90.000,B 90.000,C 0.000} C_DIS
LIN {X -4.092,Y -46.965,Z -132.722,A -90.000,B 90.000,C 0.000} C_DIS
LIN {X -4.084,Y -46.973,Z -132.596,A -90.000,B 90.000,C 0.000} C_DIS
LIN {X -4.068,Y -46.983,Z -132.383,A -90.000,B 90.000,C 0.000} C_DIS
LIN {X -4.049,Y -46.983,Z -132.146,A -90.000,B 90.000,C 0.000} C_DIS
LIN {X -3.875,Y -46.929,Z -130.138,A -90.000,B 90.000,C 0.000} C_DIS
LIN {X -3.841,Y -46.926,Z -129.904,A -90.000,B 90.000,C 0.000} C_DIS
LIN {X -3.684,Y -46.923,Z -129.137,A -90.000,B 90.000,C 0.000} C_DIS
LIN {X -3.657,Y -46.923,Z -129.023,A -90.000,B 90.000,C 0.000} C_DIS
LIN {X -3.587,Y -46.926,Z -128.788,A -90.000,B 90.000,C 0.000} C_DIS
LIN {X -3.556,Y -46.927,Z -128.699,A -90.000,B 90.000,C 0.000} C_DIS
LIN {X -3.502,Y -46.930,Z -128.569,A -90.000,B 90.000,C 0.000} C_DIS
LIN {X -3.438,Y -46.929,Z -128.441,A -90.000,B 90.000,C 0.000} C_DIS
LIN {X -3.316,Y -46.929,Z -128.221,A -90.000,B 90.000,C 0.000} C_DIS
LIN {X -3.144,Y -46.930,Z -127.921,A -90.000,B 90.000,C 0.000} C_DIS
LIN {X -3.096,Y -46.930,Z -127.841,A -90.000,B 90.000,C 0.000} C_DIS
LIN {X -2.137,Y -46.952,Z -126.335,A -90.000,B 90.000,C 0.000} C_DIS
LIN {X -1.852,Y -46.955,Z -125.888,A -90.000,B 90.000,C 0.000} C_DIS
LIN {X -1.602,Y -46.955,Z -125.497,A -90.000,B 90.000,C 0.000} C_DIS
LIN {X -1.392,Y -46.947,Z -125.173,A -90.000,B 90.000,C 0.000} C_DIS
LIN {X -1.271,Y -46.946,Z -125.014,A -90.000,B 90.000,C 0.000} C_DIS
LIN {X -0.944,Y -46.946,Z -124.612,A -90.000,B 90.000,C 0.000} C_DIS
LIN {X -0.824,Y -46.947,Z -124.478,A -90.000,B 90.000,C 0.000} C_DIS
LIN {X -0.670,Y -46.951,Z -124.322,A -90.000,B 90.000,C 0.000} C_DIS
LIN {X 0.228,Y -46.978,Z -123.459,A -90.000,B 90.000,C 0.000} C_DIS
LIN {X 0.971,Y -46.979,Z -122.751,A -90.000,B 90.000,C 0.000} C_DIS
LIN {X 1.663,Y -46.984,Z -122.115,A -90.000,B 90.000,C 0.000} C_DIS
LIN {X 1.822,Y -46.987,Z -121.983,A -90.000,B 90.000,C 0.000} C_DIS
LIN {X 2.116,Y -46.995,Z -121.764,A -90.000,B 90.000,C 0.000} C_DIS
LIN {X 2.631,Y -47.013,Z -121.407,A -90.000,B 90.000,C 0.000} C_DIS
LIN {X 4.350,Y -47.014,Z -120.225,A -90.000,B 90.000,C 0.000} C_DIS
LIN {X 4.494,Y -47.015,Z -120.134,A -90.000,B 90.000,C 0.000} C_DIS
LIN {X 4.649,Y -47.018,Z -120.046,A -90.000,B 90.000,C 0.000} C_DIS
LIN {X 4.791,Y -47.020,Z -119.971,A -90.000,B 90.000,C 0.000} C_DIS
LIN {X 5.500,Y -47.037,Z -119.611,A -90.000,B 90.000,C 0.000} C_DIS
LIN {X 7.542,Y -47.041,Z -118.579,A -90.000,B 90.000,C 0.000} C_DIS
LIN {X 7.857,Y -47.043,Z -118.414,A -90.000,B 90.000,C 0.000} C_DIS
LIN {X 8.109,Y -47.044,Z -118.273,A -90.000,B 90.000,C 0.000} C_DIS
LIN {X 8.407,Y -47.046,Z -118.128,A -90.000,B 90.000,C 0.000} C_DIS
LIN {X 8.811,Y -47.047,Z -117.956,A -90.000,B 90.000,C 0.000} C_DIS
LIN {X 8.970,Y -47.048,Z -117.884,A -90.000,B 90.000,C 0.000} C_DIS
LIN {X 9.287,Y -47.049,Z -117.734,A -90.000,B 90.000,C 0.000} C_DIS
LIN {X 9.600,Y -47.050,Z -117.578,A -90.000,B 90.000,C 0.000} C_DIS
LIN {X 10.064,Y -47.048,Z -117.331,A -90.000,B 90.000,C 0.000} C_DIS
LIN {X 10.370,Y -47.046,Z -117.160,A -90.000,B 90.000,C 0.000} C_DIS
LIN {X 10.674,Y -47.043,Z -116.985,A -90.000,B 90.000,C 0.000} C_DIS
LIN {X 11.276,Y -47.039,Z -116.623,A -90.000,B 90.000,C 0.000} C_DIS
LIN {X 11.873,Y -47.034,Z -116.251,A -90.000,B 90.000,C 0.000} C_DIS
LIN {X 12.763,Y -47.027,Z -115.684,A -90.000,B 90.000,C 0.000} C_DIS
LIN {X 13.062,Y -47.025,Z -115.501,A -90.000,B 90.000,C 0.000} C_DIS
LIN {X 13.251,Y -47.024,Z -115.396,A -90.000,B 90.000,C 0.000} C_DIS
LIN {X 13.442,Y -47.022,Z -115.302,A -90.000,B 90.000,C 0.000} C_DIS
LIN {X 13.752,Y -47.020,Z -115.160,A -90.000,B 90.000,C 0.000} C_DIS
LIN {X 13.868,Y -47.019,Z -115.111,A -90.000,B 90.000,C 0.000} C_DIS
LIN {X 13.986,Y -47.018,Z -115.068,A -90.000,B 90.000,C 0.000} C_DIS
LIN {X 14.459,Y -47.015,Z -114.897,A -90.000,B 90.000,C 0.000} C_DIS
LIN {X 14.777,Y -47.013,Z -114.787,A -90.000,B 90.000,C 0.000} C_DIS
LIN {X 15.259,Y -47.010,Z -114.632,A -90.000,B 90.000,C 0.000} C_DIS
LIN {X 15.747,Y -47.006,Z -114.492,A -90.000,B 90.000,C 0.000} C_DIS
LIN {X 16.078,Y -47.004,Z -114.407,A -90.000,B 90.000,C 0.000} C_DIS
LIN {X 16.244,Y -47.003,Z -114.368,A -90.000,B 90.000,C 0.000} C_DIS
LIN {X 16.580,Y -47.001,Z -114.295,A -90.000,B 90.000,C 0.000} C_DIS
LIN {X 16.750,Y -47.000,Z -114.262,A -90.000,B 90.000,C 0.000} C_DIS
LIN {X 17.093,Y -46.997,Z -114.204,A -90.000,B 90.000,C 0.000} C_DIS
LIN {X 17.266,Y -46.996,Z -114.178,A -90.000,B 90.000,C 0.000} C_DIS
LIN {X 17.616,Y -46.993,Z -114.135,A -90.000,B 90.000,C 0.000} C_DIS
LIN {X 18.015,Y -46.994,Z -114.094,A -90.000,B 90.000,C 0.000} C_DIS
LIN {X 18.135,Y -46.995,Z -114.085,A -90.000,B 90.000,C 0.000} C_DIS
LIN {X 18.311,Y -46.996,Z -114.077,A -90.000,B 90.000,C 0.000} C_DIS
LIN {X 18.793,Y -47.000,Z -114.075,A -90.000,B 90.000,C 0.000} C_DIS
LIN {X 18.916,Y -47.002,Z -114.078,A -90.000,B 90.000,C 0.000} C_DIS
LIN {X 19.286,Y -47.007,Z -114.110,A -90.000,B 90.000,C 0.000} C_DIS
LIN {X 19.488,Y -47.011,Z -114.135,A -90.000,B 90.000,C 0.000} C_DIS
LIN {X 20.051,Y -47.023,Z -114.234,A -90.000,B 90.000,C 0.000} C_DIS
LIN {X 21.364,Y -47.054,Z -114.465,A -90.000,B 90.000,C 0.000} C_DIS
LIN {X 22.684,Y -47.058,Z -114.699,A -90.000,B 90.000,C 0.000} C_DIS
LIN {X 23.436,Y -47.062,Z -114.850,A -90.000,B 90.000,C 0.000} C_DIS
LIN {X 23.543,Y -47.062,Z -114.875,A -90.000,B 90.000,C 0.000} C_DIS
LIN {X 23.862,Y -47.065,Z -114.964,A -90.000,B 90.000,C 0.000} C_DIS
LIN {X 24.054,Y -47.068,Z -115.028,A -90.000,B 90.000,C 0.000} C_DIS
LIN {X 24.157,Y -47.069,Z -115.072,A -90.000,B 90.000,C 0.000} C_DIS
LIN {X 24.522,Y -47.077,Z -115.241,A -90.000,B 90.000,C 0.000} C_DIS
LIN {X 24.680,Y -47.081,Z -115.329,A -90.000,B 90.000,C 0.000} C_DIS
LIN {X 24.887,Y -47.087,Z -115.459,A -90.000,B 90.000,C 0.000} C_DIS
LIN {X 24.947,Y -47.089,Z -115.502,A -90.000,B 90.000,C 0.000} C_DIS
LIN {X 25.073,Y -47.091,Z -115.594,A -90.000,B 90.000,C 0.000} C_DIS
LIN {X 26.732,Y -47.091,Z -116.885,A -90.000,B 90.000,C 0.000} C_DIS
LIN {X 27.044,Y -47.091,Z -117.131,A -90.000,B 90.000,C 0.000} C_DIS
LIN {X 27.126,Y -47.091,Z -117.201,A -90.000,B 90.000,C 0.000} C_DIS
LIN {X 27.241,Y -47.091,Z -117.302,A -90.000,B 90.000,C 0.000} C_DIS
LIN {X 27.384,Y -47.091,Z -117.438,A -90.000,B 90.000,C 0.000} C_DIS
LIN {X 27.454,Y -47.091,Z -117.508,A -90.000,B 90.000,C 0.000} C_DIS
LIN {X 27.533,Y -47.092,Z -117.593,A -90.000,B 90.000,C 0.000} C_DIS
LIN {X 27.801,Y -47.093,Z -117.895,A -90.000,B 90.000,C 0.000} C_DIS
LIN {X 28.269,Y -47.068,Z -118.428,A -90.000,B 90.000,C 0.000} C_DIS
LIN {X 28.360,Y -47.063,Z -118.536,A -90.000,B 90.000,C 0.000} C_DIS
LIN {X 28.544,Y -47.054,Z -118.774,A -90.000,B 90.000,C 0.000} C_DIS
LIN {X 28.628,Y -47.049,Z -118.895,A -90.000,B 90.000,C 0.000} C_DIS
LIN {X 28.706,Y -47.045,Z -119.020,A -90.000,B 90.000,C 0.000} C_DIS
LIN {X 28.791,Y -47.041,Z -119.166,A -90.000,B 90.000,C 0.000} C_DIS
LIN {X 28.903,Y -47.034,Z -119.385,A -90.000,B 90.000,C 0.000} C_DIS
LIN {X 28.938,Y -47.031,Z -119.461,A -90.000,B 90.000,C 0.000} C_DIS
LIN {X 29.008,Y -47.026,Z -119.632,A -90.000,B 90.000,C 0.000} C_DIS
LIN {X 29.093,Y -47.019,Z -119.872,A -90.000,B 90.000,C 0.000} C_DIS
LIN {X 29.144,Y -47.015,Z -120.036,A -90.000,B 90.000,C 0.000} C_DIS
LIN {X 29.183,Y -47.012,Z -120.180,A -90.000,B 90.000,C 0.000} C_DIS
LIN {X 29.243,Y -47.007,Z -120.449,A -90.000,B 90.000,C 0.000} C_DIS
LIN {X 29.396,Y -46.996,Z -121.316,A -90.000,B 90.000,C 0.000} C_DIS
LIN {X 29.423,Y -46.993,Z -121.469,A -90.000,B 90.000,C 0.000} C_DIS
LIN {X 29.485,Y -46.984,Z -121.841,A -90.000,B 90.000,C 0.000} C_DIS
LIN {X 29.501,Y -46.981,Z -121.972,A -90.000,B 90.000,C 0.000} C_DIS
LIN {X 29.512,Y -46.976,Z -122.094,A -90.000,B 90.000,C 0.000} C_DIS
LIN {X 29.521,Y -46.967,Z -122.267,A -90.000,B 90.000,C 0.000} C_DIS
LIN {X 29.523,Y -46.961,Z -122.386,A -90.000,B 90.000,C 0.000} C_DIS
LIN {X 29.515,Y -46.951,Z -122.617,A -90.000,B 90.000,C 0.000} C_DIS
LIN {X 29.503,Y -46.945,Z -122.774,A -90.000,B 90.000,C 0.000} C_DIS
LIN {X 29.439,Y -46.927,Z -123.335,A -90.000,B 90.000,C 0.000} C_DIS
LIN {X 29.487,Y -46.893,Z -123.933,A -90.000,B 90.000,C 0.000} C_DIS
LIN {X 29.530,Y -46.839,Z -124.523,A -90.000,B 90.000,C 0.000} C_DIS
LIN {X 29.535,Y -46.830,Z -124.627,A -90.000,B 90.000,C 0.000} C_DIS
LIN {X 29.534,Y -46.823,Z -124.713,A -90.000,B 90.000,C 0.000} C_DIS
LIN {X 29.526,Y -46.801,Z -124.994,A -90.000,B 90.000,C 0.000} C_DIS
LIN {X 29.508,Y -46.786,Z -125.212,A -90.000,B 90.000,C 0.000} C_DIS
LIN {X 29.484,Y -46.775,Z -125.382,A -90.000,B 90.000,C 0.000} C_DIS
LIN {X 29.452,Y -46.765,Z -125.587,A -90.000,B 90.000,C 0.000} C_DIS
LIN {X 29.434,Y -46.762,Z -125.689,A -90.000,B 90.000,C 0.000} C_DIS
LIN {X 29.348,Y -46.750,Z -126.072,A -90.000,B 90.000,C 0.000} C_DIS
LIN {X 29.320,Y -46.742,Z -126.192,A -90.000,B 90.000,C 0.000} C_DIS
LIN {X 28.931,Y -46.627,Z -127.866,A -90.000,B 90.000,C 0.000} C_DIS
LIN {X 28.910,Y -46.617,Z -127.950,A -90.000,B 90.000,C 0.000} C_DIS
LIN {X 28.869,Y -46.601,Z -128.099,A -90.000,B 90.000,C 0.000} C_DIS
LIN {X 28.762,Y -46.568,Z -128.434,A -90.000,B 90.000,C 0.000} C_DIS
LIN {X 28.666,Y -46.547,Z -128.682,A -90.000,B 90.000,C 0.000} C_DIS
LIN {X 28.596,Y -46.532,Z -128.846,A -90.000,B 90.000,C 0.000} C_DIS
LIN {X 28.541,Y -46.523,Z -128.960,A -90.000,B 90.000,C 0.000} C_DIS
LIN {X 28.362,Y -46.497,Z -129.310,A -90.000,B 90.000,C 0.000} C_DIS
LIN {X 28.161,Y -46.458,Z -129.697,A -90.000,B 90.000,C 0.000} C_DIS
LIN {X 27.299,Y -46.317,Z -131.371,A -90.000,B 90.000,C 0.000} C_DIS
LIN {X 26.978,Y -46.272,Z -131.964,A -90.000,B 90.000,C 0.000} C_DIS
LIN {X 26.896,Y -46.263,Z -132.105,A -90.000,B 90.000,C 0.000} C_DIS
LIN {X 26.768,Y -46.253,Z -132.308,A -90.000,B 90.000,C 0.000} C_DIS
LIN {X 26.681,Y -46.248,Z -132.430,A -90.000,B 90.000,C 0.000} C_DIS
LIN {X 26.605,Y -46.245,Z -132.535,A -90.000,B 90.000,C 0.000} C_DIS
LIN {X 26.460,Y -46.229,Z -132.729,A -90.000,B 90.000,C 0.000} C_DIS
LIN {X 25.348,Y -46.088,Z -134.302,A -90.000,B 90.000,C 0.000} C_DIS
LIN {X 25.110,Y -46.066,Z -134.644,A -90.000,B 90.000,C 0.000} C_DIS
LIN {X 25.046,Y -46.061,Z -134.731,A -90.000,B 90.000,C 0.000} C_DIS
LIN {X 24.933,Y -46.055,Z -134.876,A -90.000,B 90.000,C 0.000} C_DIS
LIN {X 24.831,Y -46.051,Z -135.000,A -90.000,B 90.000,C 0.000} C_DIS
LIN {X 24.600,Y -46.047,Z -135.269,A -90.000,B 90.000,C 0.000} C_DIS
LIN {X 24.397,Y -46.027,Z -135.493,A -90.000,B 90.000,C 0.000} C_DIS
LIN {X 24.041,Y -45.988,Z -135.883,A -90.000,B 90.000,C 0.000} C_DIS
LIN {X 23.854,Y -45.973,Z -136.070,A -90.000,B 90.000,C 0.000} C_DIS
LIN {X 23.063,Y -45.926,Z -136.817,A -90.000,B 90.000,C 0.000} C_DIS
LIN {X 22.525,Y -45.906,Z -137.334,A -90.000,B 90.000,C 0.000} C_DIS
LIN {X 22.297,Y -45.895,Z -137.550,A -90.000,B 90.000,C 0.000} C_DIS
LIN {X 22.120,Y -45.873,Z -137.711,A -90.000,B 90.000,C 0.000} C_DIS
LIN {X 21.347,Y -45.796,Z -138.369,A -90.000,B 90.000,C 0.000} C_DIS
LIN {X 21.019,Y -45.770,Z -138.632,A -90.000,B 90.000,C 0.000} C_DIS
LIN {X 20.910,Y -45.764,Z -138.713,A -90.000,B 90.000,C 0.000} C_DIS
LIN {X 20.702,Y -45.756,Z -138.859,A -90.000,B 90.000,C 0.000} C_DIS
LIN {X 20.533,Y -45.754,Z -138.966,A -90.000,B 90.000,C 0.000} C_DIS
LIN {X 20.185,Y -45.760,Z -139.167,A -90.000,B 90.000,C 0.000} C_DIS
LIN {X 19.845,Y -45.767,Z -139.350,A -90.000,B 90.000,C 0.000} C_DIS
LIN {X 19.581,Y -45.761,Z -139.484,A -90.000,B 90.000,C 0.000} C_DIS
LIN {X 18.788,Y -45.744,Z -139.879,A -90.000,B 90.000,C 0.000} C_DIS
LIN {X 18.073,Y -45.727,Z -140.238,A -90.000,B 90.000,C 0.000} C_DIS
LIN {X 17.336,Y -45.688,Z -140.600,A -90.000,B 90.000,C 0.000} C_DIS
LIN {X 16.939,Y -45.669,Z -140.793,A -90.000,B 90.000,C 0.000} C_DIS
LIN {X 16.607,Y -45.644,Z -140.949,A -90.000,B 90.000,C 0.000} C_DIS
LIN {X 16.377,Y -45.619,Z -141.052,A -90.000,B 90.000,C 0.000} C_DIS
LIN {X 16.265,Y -45.609,Z -141.099,A -90.000,B 90.000,C 0.000} C_DIS
LIN {X 16.044,Y -45.593,Z -141.185,A -90.000,B 90.000,C 0.000} C_DIS
LIN {X 15.930,Y -45.587,Z -141.226,A -90.000,B 90.000,C 0.000} C_DIS
LIN {X 15.721,Y -45.579,Z -141.295,A -90.000,B 90.000,C 0.000} C_DIS
LIN {X 15.080,Y -45.561,Z -141.498,A -90.000,B 90.000,C 0.000} C_DIS
LIN {X 14.928,Y -45.559,Z -141.543,A -90.000,B 90.000,C 0.000} C_DIS
LIN {X 14.788,Y -45.558,Z -141.581,A -90.000,B 90.000,C 0.000} C_DIS
LIN {X 14.699,Y -45.558,Z -141.605,A -90.000,B 90.000,C 0.000} C_DIS
LIN {X 14.515,Y -45.560,Z -141.648,A -90.000,B 90.000,C 0.000} C_DIS
LIN {X 14.332,Y -45.565,Z -141.687,A -90.000,B 90.000,C 0.000} C_DIS
LIN {X 13.252,Y -45.611,Z -141.884,A -90.000,B 90.000,C 0.000} C_DIS
LIN {X 12.975,Y -45.626,Z -141.931,A -90.000,B 90.000,C 0.000} C_DIS
LIN {X 12.634,Y -45.636,Z -141.981,A -90.000,B 90.000,C 0.000} C_DIS
LIN {X 11.689,Y -45.641,Z -142.108,A -90.000,B 90.000,C 0.000} C_DIS
LIN {X 10.198,Y -45.648,Z -142.311,A -90.000,B 90.000,C 0.000} C_DIS
LIN {X 10.053,Y -45.651,Z -142.326,A -90.000,B 90.000,C 0.000} C_DIS
LIN {X 9.787,Y -45.661,Z -142.347,A -90.000,B 90.000,C 0.000} C_DIS
LIN {X 9.654,Y -45.668,Z -142.353,A -90.000,B 90.000,C 0.000} C_DIS
LIN {X 9.347,Y -45.690,Z -142.359,A -90.000,B 90.000,C 0.000} C_DIS
LIN {X 8.485,Y -45.741,Z -142.373,A -90.000,B 90.000,C 0.000} C_DIS
LIN {X 8.160,Y -45.750,Z -142.374,A -90.000,B 90.000,C 0.000} C_DIS
LIN {X 6.951,Y -45.753,Z -142.363,A -90.000,B 90.000,C 0.000} C_DIS
LIN {X 5.762,Y -45.764,Z -142.338,A -90.000,B 90.000,C 0.000} C_DIS
LIN {X 5.670,Y -45.766,Z -142.334,A -90.000,B 90.000,C 0.000} C_DIS
LIN {X 5.173,Y -45.781,Z -142.303,A -90.000,B 90.000,C 0.000} C_DIS
LIN {X 5.070,Y -45.786,Z -142.294,A -90.000,B 90.000,C 0.000} C_DIS
LIN {X 4.866,Y -45.797,Z -142.272,A -90.000,B 90.000,C 0.000} C_DIS
LIN {X 4.776,Y -45.803,Z -142.261,A -90.000,B 90.000,C 0.000} C_DIS
LIN {X 4.448,Y -45.829,Z -142.211,A -90.000,B 90.000,C 0.000} C_DIS
LIN {X 4.288,Y -45.846,Z -142.179,A -90.000,B 90.000,C 0.000} C_DIS
LIN {X 4.154,Y -45.858,Z -142.148,A -90.000,B 90.000,C 0.000} C_DIS
LIN {X 3.926,Y -45.882,Z -142.082,A -90.000,B 90.000,C 0.000} C_DIS
LIN {X 3.545,Y -45.915,Z -141.946,A -90.000,B 90.000,C 0.000} C_DIS
LIN {X 2.619,Y -45.963,Z -141.676,A -90.000,B 90.000,C 0.000} C_DIS
LIN {X 0.736,Y -46.039,Z -141.116,A -90.000,B 90.000,C 0.000} C_DIS
LIN {X 0.677,Y -46.042,Z -141.097,A -90.000,B 90.000,C 0.000} C_DIS
LIN {X 0.521,Y -46.051,Z -141.043,A -90.000,B 90.000,C 0.000} C_DIS
LIN {X 0.231,Y -46.073,Z -140.931,A -90.000,B 90.000,C 0.000} C_DIS
LIN {X 0.080,Y -46.085,Z -140.868,A -90.000,B 90.000,C 0.000} C_DIS
LIN {X 0.010,Y -46.087,Z -140.835,A -90.000,B 90.000,C 0.000} C_DIS
LIN {X -0.117,Y -46.093,Z -140.771,A -90.000,B 90.000,C 0.000} C_DIS
LIN {X -0.236,Y -46.098,Z -140.705,A -90.000,B 90.000,C 0.000} C_DIS
LIN {X -0.449,Y -46.113,Z -140.575,A -90.000,B 90.000,C 0.000} C_DIS
LIN {X -0.719,Y -46.128,Z -140.393,A -90.000,B 90.000,C 0.000} C_DIS
LIN {X -0.913,Y -46.142,Z -140.251,A -90.000,B 90.000,C 0.000} C_DIS
LIN {X -1.013,Y -46.151,Z -140.168,A -90.000,B 90.000,C 0.000} C_DIS
LIN {X -2.139,Y -46.269,Z -139.210,A -90.000,B 90.000,C 0.000} C_DIS
LIN {X -2.887,Y -46.333,Z -138.625,A -90.000,B 90.000,C 0.000} C_DIS
LIN {X -3.132,Y -46.346,Z -138.431,A -90.000,B 90.000,C 0.000} C_DIS
LIN {X -3.427,Y -46.339,Z -138.190,A -90.000,B 90.000,C 0.000} C_DIS
LIN {X -3.582,Y -46.335,Z -138.058,A -90.000,B 90.000,C 0.000} C_DIS
LIN {X -3.710,Y -46.334,Z -137.938,A -90.000,B 90.000,C 0.000} C_DIS
LIN {X -3.806,Y -46.334,Z -137.841,A -90.000,B 90.000,C 0.000} C_DIS
LIN {X -3.971,Y -46.336,Z -137.670,A -90.000,B 90.000,C 0.000} C_DIS
LIN {X -4.169,Y -46.343,Z -137.448,A -90.000,B 90.000,C 0.000} C_DIS
LIN {X -4.219,Y -46.345,Z -137.388,A -90.000,B 90.000,C 0.000} C_DIS
LIN {X -4.297,Y -46.351,Z -137.286,A -90.000,B 90.000,C 0.000} C_DIS
LIN {X -4.441,Y -46.365,Z -137.084,A -90.000,B 90.000,C 0.000} C_DIS
LIN {X -4.594,Y -46.385,Z -136.846,A -90.000,B 90.000,C 0.000} C_DIS
LIN {X -4.716,Y -46.403,Z -136.646,A -90.000,B 90.000,C 0.000} C_DIS
LIN {X -4.913,Y -46.438,Z -136.298,A -90.000,B 90.000,C 0.000} C_DIS
LIN {X -5.275,Y -46.492,Z -135.653,A -90.000,B 90.000,C 0.000} C_DIS
LIN {X -5.380,Y -46.494,Z -135.458,A -90.000,B 90.000,C 0.000} C_DIS
LIN {X -5.442,Y -46.496,Z -135.335,A -90.000,B 90.000,C 0.000} C_DIS
LIN {X -5.498,Y -46.498,Z -135.212,A -90.000,B 90.000,C 0.000} C_DIS
LIN {X -5.546,Y -46.496,Z -135.100,A -90.000,B 90.000,C 0.000} C_DIS
LIN {X -5.574,Y -46.496,Z -135.026,A -90.000,B 90.000,C 0.000} C_DIS
LIN {X -5.584,Y -46.495,Z -134.999,A -90.000,B 90.000,C 0.000} C_DIS
LIN {X -5.802,Y -46.474,Z -134.378,A -90.000,B 90.000,C 0.000} C_DIS
LIN {X -5.855,Y -46.470,Z -134.200,A -90.000,B 90.000,C 0.000} C_DIS
LIN {X -5.944,Y -46.467,Z -133.845,A -90.000,B 90.000,C 0.000} C_DIS
LIN {X -5.985,Y -46.467,Z -133.633,A -90.000,B 90.000,C 0.000} C_DIS
LIN {X -6.008,Y -46.471,Z -133.459,A -90.000,B 90.000,C 0.000} C_DIS
LIN {X -6.016,Y -46.473,Z -133.364,A -90.000,B 90.000,C 0.000} C_DIS
LIN {X -6.038,Y -46.485,Z -133.032,A -90.000,B 90.000,C 0.000} C_DIS
LIN {X -6.038,Y -46.501,Z -132.704,A -90.000,B 90.000,C 0.000} C_DIS
LIN {X -6.036,Y -46.506,Z -132.606,A -90.000,B 90.000,C 0.000} C_DIS
LIN {X -5.975,Y -46.566,Z -131.703,A -90.000,B 90.000,C 0.000} C_DIS
LIN {X -5.961,Y -46.575,Z -131.506,A -90.000,B 90.000,C 0.000} C_DIS
LIN {X -5.943,Y -46.575,Z -131.287,A -90.000,B 90.000,C 0.000} C_DIS
LIN {X -5.831,Y -46.542,Z -129.980,A -90.000,B 90.000,C 0.000} C_DIS
LIN {X -5.817,Y -46.539,Z -129.862,A -90.000,B 90.000,C 0.000} C_DIS
LIN {X -5.771,Y -46.530,Z -129.558,A -90.000,B 90.000,C 0.000} C_DIS
LIN {X -5.600,Y -46.508,Z -128.745,A -90.000,B 90.000,C 0.000} C_DIS
LIN {X -5.560,Y -46.505,Z -128.574,A -90.000,B 90.000,C 0.000} C_DIS
LIN {X -5.529,Y -46.503,Z -128.461,A -90.000,B 90.000,C 0.000} C_DIS
LIN {X -5.501,Y -46.503,Z -128.364,A -90.000,B 90.000,C 0.000} C_DIS
LIN {X -5.434,Y -46.505,Z -128.146,A -90.000,B 90.000,C 0.000} C_DIS
LIN {X -5.370,Y -46.508,Z -127.968,A -90.000,B 90.000,C 0.000} C_DIS
LIN {X -5.285,Y -46.513,Z -127.763,A -90.000,B 90.000,C 0.000} C_DIS
LIN {X -5.258,Y -46.516,Z -127.706,A -90.000,B 90.000,C 0.000} C_DIS
LIN {X -5.180,Y -46.514,Z -127.551,A -90.000,B 90.000,C 0.000} C_DIS
LIN {X -5.033,Y -46.512,Z -127.284,A -90.000,B 90.000,C 0.000} C_DIS
LIN {X -4.840,Y -46.512,Z -126.947,A -90.000,B 90.000,C 0.000} C_DIS
LIN {X -4.743,Y -46.513,Z -126.786,A -90.000,B 90.000,C 0.000} C_DIS
LIN {X -4.042,Y -46.526,Z -125.686,A -90.000,B 90.000,C 0.000} C_DIS
LIN {X -3.526,Y -46.556,Z -124.868,A -90.000,B 90.000,C 0.000} C_DIS
LIN {X -3.350,Y -46.561,Z -124.591,A -90.000,B 90.000,C 0.000} C_DIS
LIN {X -3.064,Y -46.550,Z -124.150,A -90.000,B 90.000,C 0.000} C_DIS
LIN {X -2.986,Y -46.548,Z -124.033,A -90.000,B 90.000,C 0.000} C_DIS
LIN {X -2.790,Y -46.546,Z -123.775,A -90.000,B 90.000,C 0.000} C_DIS
LIN {X -2.490,Y -46.548,Z -123.407,A -90.000,B 90.000,C 0.000} C_DIS
LIN {X -2.405,Y -46.548,Z -123.305,A -90.000,B 90.000,C 0.000} C_DIS
LIN {X -2.284,Y -46.551,Z -123.170,A -90.000,B 90.000,C 0.000} C_DIS
LIN {X -2.216,Y -46.552,Z -123.097,A -90.000,B 90.000,C 0.000} C_DIS
LIN {X -2.063,Y -46.558,Z -122.941,A -90.000,B 90.000,C 0.000} C_DIS
LIN {X -1.768,Y -46.569,Z -122.656,A -90.000,B 90.000,C 0.000} C_DIS
LIN {X -0.962,Y -46.624,Z -121.875,A -90.000,B 90.000,C 0.000} C_DIS
LIN {X -0.388,Y -46.631,Z -121.325,A -90.000,B 90.000,C 0.000} C_DIS
LIN {X 0.331,Y -46.642,Z -120.663,A -90.000,B 90.000,C 0.000} C_DIS
LIN {X 0.409,Y -46.643,Z -120.595,A -90.000,B 90.000,C 0.000} C_DIS
LIN {X 0.567,Y -46.648,Z -120.463,A -90.000,B 90.000,C 0.000} C_DIS
LIN {X 0.653,Y -46.651,Z -120.395,A -90.000,B 90.000,C 0.000} C_DIS
LIN {X 0.995,Y -46.664,Z -120.142,A -90.000,B 90.000,C 0.000} C_DIS
LIN {X 1.825,Y -46.701,Z -119.564,A -90.000,B 90.000,C 0.000} C_DIS
LIN {X 2.274,Y -46.717,Z -119.252,A -90.000,B 90.000,C 0.000} C_DIS
LIN {X 3.229,Y -46.719,Z -118.595,A -90.000,B 90.000,C 0.000} C_DIS
LIN {X 3.443,Y -46.723,Z -118.458,A -90.000,B 90.000,C 0.000} C_DIS
LIN {X 3.672,Y -46.727,Z -118.325,A -90.000,B 90.000,C 0.000} C_DIS
LIN {X 3.812,Y -46.730,Z -118.250,A -90.000,B 90.000,C 0.000} C_DIS
LIN {X 6.939,Y -46.810,Z -116.659,A -90.000,B 90.000,C 0.000} C_DIS
LIN {X 7.217,Y -46.814,Z -116.518,A -90.000,B 90.000,C 0.000} C_DIS
LIN {X 7.369,Y -46.817,Z -116.448,A -90.000,B 90.000,C 0.000} C_DIS
LIN {X 7.674,Y -46.825,Z -116.325,A -90.000,B 90.000,C 0.000} C_DIS
LIN {X 7.820,Y -46.829,Z -116.272,A -90.000,B 90.000,C 0.000} C_DIS
LIN {X 10.276,Y -46.865,Z -115.510,A -90.000,B 90.000,C 0.000} C_DIS
LIN {X 12.728,Y -46.906,Z -114.750,A -90.000,B 90.000,C 0.000} C_DIS
LIN {X 12.889,Y -46.907,Z -114.705,A -90.000,B 90.000,C 0.000} C_DIS
LIN {X 13.132,Y -46.907,Z -114.645,A -90.000,B 90.000,C 0.000} C_DIS
LIN {X 13.265,Y -46.910,Z -114.617,A -90.000,B 90.000,C 0.000} C_DIS
LIN {X 13.503,Y -46.913,Z -114.573,A -90.000,B 90.000,C 0.000} C_DIS
LIN {X 13.600,Y -46.914,Z -114.559,A -90.000,B 90.000,C 0.000} C_DIS
LIN {X 13.958,Y -46.920,Z -114.525,A -90.000,B 90.000,C 0.000} C_DIS
LIN {X 17.546,Y -46.993,Z -114.143,A -90.000,B 90.000,C 0.000} C_DIS
LIN {X 17.616,Y -46.993,Z -114.135,A -90.000,B 90.000,C 0.000} C_DIS
LIN {X 17.616,Y -60.000,Z -114.135,A -90.000,B 90.000,C 0.000} C_DIS
LIN {X -1.622,Y -60.000,Z -141.989,A -90.000,B 90.000,C 0.000} C_DIS
LIN {X -1.622,Y -45.308,Z -141.989,A -90.000,B 90.000,C 0.000} C_DIS
LIN {X -1.783,Y -45.325,Z -141.884,A -90.000,B 90.000,C 0.000} C_DIS
LIN {X -2.038,Y -45.358,Z -141.707,A -90.000,B 90.000,C 0.000} C_DIS
LIN {X -2.130,Y -45.372,Z -141.639,A -90.000,B 90.000,C 0.000} C_DIS
LIN {X -2.285,Y -45.398,Z -141.516,A -90.000,B 90.000,C 0.000} C_DIS
LIN {X -2.958,Y -45.518,Z -140.969,A -90.000,B 90.000,C 0.000} C_DIS
LIN {X -3.368,Y -45.595,Z -140.637,A -90.000,B 90.000,C 0.000} C_DIS
LIN {X -3.703,Y -45.649,Z -140.386,A -90.000,B 90.000,C 0.000} C_DIS
LIN {X -3.956,Y -45.682,Z -140.194,A -90.000,B 90.000,C 0.000} C_DIS
LIN {X -4.216,Y -45.696,Z -139.988,A -90.000,B 90.000,C 0.000} C_DIS
LIN {X -4.645,Y -45.711,Z -139.646,A -90.000,B 90.000,C 0.000} C_DIS
LIN {X -4.827,Y -45.719,Z -139.497,A -90.000,B 90.000,C 0.000} C_DIS
LIN {X -5.058,Y -45.734,Z -139.289,A -90.000,B 90.000,C 0.000} C_DIS
LIN {X -5.300,Y -45.757,Z -139.051,A -90.000,B 90.000,C 0.000} C_DIS
LIN {X -5.412,Y -45.762,Z -138.934,A -90.000,B 90.000,C 0.000} C_DIS
LIN {X -5.609,Y -45.773,Z -138.713,A -90.000,B 90.000,C 0.000} C_DIS
LIN {X -5.732,Y -45.782,Z -138.569,A -90.000,B 90.000,C 0.000} C_DIS
LIN {X -5.853,Y -45.794,Z -138.412,A -90.000,B 90.000,C 0.000} C_DIS
LIN {X -6.024,Y -45.812,Z -138.174,A -90.000,B 90.000,C 0.000} C_DIS
LIN {X -6.156,Y -45.830,Z -137.975,A -90.000,B 90.000,C 0.000} C_DIS
LIN {X -6.270,Y -45.846,Z -137.795,A -90.000,B 90.000,C 0.000} C_DIS
LIN {X -6.423,Y -45.870,Z -137.541,A -90.000,B 90.000,C 0.000} C_DIS
LIN {X -6.560,Y -45.894,Z -137.299,A -90.000,B 90.000,C 0.000} C_DIS
LIN {X -6.651,Y -45.907,Z -137.137,A -90.000,B 90.000,C 0.000} C_DIS
LIN {X -6.801,Y -45.917,Z -136.862,A -90.000,B 90.000,C 0.000} C_DIS
LIN {X -7.071,Y -45.922,Z -136.360,A -90.000,B 90.000,C 0.000} C_DIS
LIN {X -7.155,Y -45.924,Z -136.195,A -90.000,B 90.000,C 0.000} C_DIS
LIN {X -7.259,Y -45.931,Z -135.971,A -90.000,B 90.000,C 0.000} C_DIS
LIN {X -7.308,Y -45.934,Z -135.860,A -90.000,B 90.000,C 0.000} C_DIS
LIN {X -7.378,Y -45.942,Z -135.689,A -90.000,B 90.000,C 0.000} C_DIS
LIN {X -7.625,Y -45.976,Z -135.032,A -90.000,B 90.000,C 0.000} C_DIS
LIN {X -7.670,Y -45.984,Z -134.899,A -90.000,B 90.000,C 0.000} C_DIS
LIN {X -7.724,Y -45.994,Z -134.727,A -90.000,B 90.000,C 0.000} C_DIS
LIN {X -7.836,Y -46.023,Z -134.319,A -90.000,B 90.000,C 0.000} C_DIS
LIN {X -7.872,Y -46.028,Z -134.153,A -90.000,B 90.000,C 0.000} C_DIS
LIN {X -7.910,Y -46.030,Z -133.959,A -90.000,B 90.000,C 0.000} C_DIS
LIN {X -7.945,Y -46.034,Z -133.696,A -90.000,B 90.000,C 0.000} C_DIS
LIN {X -7.961,Y -46.038,Z -133.530,A -90.000,B 90.000,C 0.000} C_DIS
LIN {X -7.988,Y -46.050,Z -133.126,A -90.000,B 90.000,C 0.000} C_DIS
LIN {X -7.991,Y -46.054,Z -133.010,A -90.000,B 90.000,C 0.000} C_DIS
LIN {X -7.990,Y -46.061,Z -132.788,A -90.000,B 90.000,C 0.000} C_DIS
LIN {X -7.985,Y -46.063,Z -132.539,A -90.000,B 90.000,C 0.000} C_DIS
LIN {X -7.976,Y -46.067,Z -132.392,A -90.000,B 90.000,C 0.000} C_DIS
LIN {X -7.895,Y -46.092,Z -131.346,A -90.000,B 90.000,C 0.000} C_DIS
LIN {X -7.807,Y -46.092,Z -130.245,A -90.000,B 90.000,C 0.000} C_DIS
LIN {X -7.766,Y -46.069,Z -129.799,A -90.000,B 90.000,C 0.000} C_DIS
LIN {X -7.739,Y -46.059,Z -129.583,A -90.000,B 90.000,C 0.000} C_DIS
LIN {X -7.679,Y -46.044,Z -129.206,A -90.000,B 90.000,C 0.000} C_DIS
LIN {X -7.545,Y -46.031,Z -128.561,A -90.000,B 90.000,C 0.000} C_DIS
LIN {X -7.486,Y -46.026,Z -128.283,A -90.000,B 90.000,C 0.000} C_DIS
LIN {X -7.436,Y -46.024,Z -128.072,A -90.000,B 90.000,C 0.000} C_DIS
LIN {X -7.387,Y -46.024,Z -127.896,A -90.000,B 90.000,C 0.000} C_DIS
LIN {X -7.301,Y -46.025,Z -127.613,A -90.000,B 90.000,C 0.000} C_DIS
LIN {X -7.259,Y -46.026,Z -127.485,A -90.000,B 90.000,C 0.000} C_DIS
LIN {X -7.173,Y -46.031,Z -127.246,A -90.000,B 90.000,C 0.000} C_DIS
LIN {X -7.059,Y -46.039,Z -126.971,A -90.000,B 90.000,C 0.000} C_DIS
LIN {X -6.987,Y -46.045,Z -126.817,A -90.000,B 90.000,C 0.000} C_DIS
LIN {X -6.958,Y -46.047,Z -126.759,A -90.000,B 90.000,C 0.000} C_DIS
LIN {X -6.875,Y -46.047,Z -126.598,A -90.000,B 90.000,C 0.000} C_DIS
LIN {X -6.718,Y -46.052,Z -126.308,A -90.000,B 90.000,C 0.000} C_DIS
LIN {X -6.497,Y -46.062,Z -125.921,A -90.000,B 90.000,C 0.000} C_DIS
LIN {X -6.385,Y -46.067,Z -125.735,A -90.000,B 90.000,C 0.000} C_DIS
LIN {X -5.304,Y -46.125,Z -124.023,A -90.000,B 90.000,C 0.000} C_DIS
LIN {X -5.228,Y -46.133,Z -123.901,A -90.000,B 90.000,C 0.000} C_DIS
LIN {X -4.981,Y -46.138,Z -123.513,A -90.000,B 90.000,C 0.000} C_DIS
LIN {X -4.687,Y -46.141,Z -123.056,A -90.000,B 90.000,C 0.000} C_DIS
LIN {X -4.619,Y -46.142,Z -122.952,A -90.000,B 90.000,C 0.000} C_DIS
LIN {X -4.546,Y -46.144,Z -122.848,A -90.000,B 90.000,C 0.000} C_DIS
LIN {X -4.351,Y -46.152,Z -122.589,A -90.000,B 90.000,C 0.000} C_DIS
LIN {X -3.951,Y -46.172,Z -122.092,A -90.000,B 90.000,C 0.000} C_DIS
LIN {X -3.869,Y -46.176,Z -121.995,A -90.000,B 90.000,C 0.000} C_DIS
LIN {X -3.682,Y -46.188,Z -121.785,A -90.000,B 90.000,C 0.000} C_DIS
LIN {X -3.537,Y -46.197,Z -121.634,A -90.000,B 90.000,C 0.000} C_DIS
LIN {X -3.424,Y -46.205,Z -121.519,A -90.000,B 90.000,C 0.000} C_DIS
LIN {X -2.886,Y -46.243,Z -120.995,A -90.000,B 90.000,C 0.000} C_DIS
LIN {X -2.053,Y -46.288,Z -120.190,A -90.000,B 90.000,C 0.000} C_DIS
LIN {X -1.722,Y -46.300,Z -119.872,A -90.000,B 90.000,C 0.000} C_DIS
LIN {X -0.967,Y -46.332,Z -119.173,A -90.000,B 90.000,C 0.000} C_DIS
LIN {X -0.839,Y -46.338,Z -119.062,A -90.000,B 90.000,C 0.000} C_DIS
LIN {X -0.650,Y -46.347,Z -118.905,A -90.000,B 90.000,C 0.000} C_DIS
LIN {X -0.517,Y -46.354,Z -118.801,A -90.000,B 90.000,C 0.000} C_DIS
LIN {X -0.127,Y -46.376,Z -118.512,A -90.000,B 90.000,C 0.000} C_DIS
LIN {X 0.114,Y -46.390,Z -118.343,A -90.000,B 90.000,C 0.000} C_DIS
LIN {X 1.466,Y -46.429,Z -117.406,A -90.000,B 90.000,C 0.000} C_DIS
LIN {X 2.165,Y -46.449,Z -116.923,A -90.000,B 90.000,C 0.000} C_DIS
LIN {X 2.379,Y -46.456,Z -116.786,A -90.000,B 90.000,C 0.000} C_DIS
LIN {X 2.566,Y -46.464,Z -116.675,A -90.000,B 90.000,C 0.000} C_DIS
LIN {X 2.738,Y -46.472,Z -116.575,A -90.000,B 90.000,C 0.000} C_DIS
LIN {X 2.917,Y -46.482,Z -116.479,A -90.000,B 90.000,C 0.000} C_DIS
LIN {X 4.060,Y -46.542,Z -115.893,A -90.000,B 90.000,C 0.000} C_DIS
LIN {X 4.583,Y -46.561,Z -115.626,A -90.000,B 90.000,C 0.000} C_DIS
LIN {X 6.338,Y -46.593,Z -114.735,A -90.000,B 90.000,C 0.000} C_DIS
LIN {X 6.549,Y -46.597,Z -114.638,A -90.000,B 90.000,C 0.000} C_DIS
LIN {X 6.626,Y -46.599,Z -114.604,A -90.000,B 90.000,C 0.000} C_DIS
LIN {X 6.997,Y -46.608,Z -114.455,A -90.000,B 90.000,C 0.000} C_DIS
LIN {X 7.143,Y -46.612,Z -114.402,A -90.000,B 90.000,C 0.000} C_DIS
LIN {X 7.234,Y -46.614,Z -114.371,A -90.000,B 90.000,C 0.000} C_DIS
LIN {X 9.803,Y -46.690,Z -113.571,A -90.000,B 90.000,C 0.000} C_DIS
LIN {X 10.385,Y -46.706,Z -113.390,A -90.000,B 90.000,C 0.000} C_DIS
LIN {X 12.023,Y -46.730,Z -112.883,A -90.000,B 90.000,C 0.000} C_DIS
LIN {X 12.344,Y -46.735,Z -112.788,A -90.000,B 90.000,C 0.000} C_DIS
LIN {X 12.652,Y -46.741,Z -112.710,A -90.000,B 90.000,C 0.000} C_DIS
LIN {X 12.907,Y -46.746,Z -112.656,A -90.000,B 90.000,C 0.000} C_DIS
LIN {X 13.218,Y -46.753,Z -112.600,A -90.000,B 90.000,C 0.000} C_DIS
LIN {X 13.327,Y -46.756,Z -112.584,A -90.000,B 90.000,C 0.000} C_DIS
LIN {X 13.434,Y -46.759,Z -112.572,A -90.000,B 90.000,C 0.000} C_DIS
LIN {X 13.761,Y -46.770,Z -112.541,A -90.000,B 90.000,C 0.000} C_DIS
LIN {X 14.915,Y -46.806,Z -112.417,A -90.000,B 90.000,C 0.000} C_DIS
LIN {X 16.670,Y -46.834,Z -112.230,A -90.000,B 90.000,C 0.000} C_DIS
LIN {X 17.716,Y -46.862,Z -112.118,A -90.000,B 90.000,C 0.000} C_DIS
LIN {X 17.987,Y -46.869,Z -112.094,A -90.000,B 90.000,C 0.000} C_DIS
LIN {X 18.135,Y -46.874,Z -112.086,A -90.000,B 90.000,C 0.000} C_DIS
LIN {X 18.313,Y -46.879,Z -112.080,A -90.000,B 90.000,C 0.000} C_DIS
LIN {X 18.855,Y -46.896,Z -112.078,A -90.000,B 90.000,C 0.000} C_DIS
LIN {X 19.033,Y -46.900,Z -112.084,A -90.000,B 90.000,C 0.000} C_DIS
LIN {X 19.457,Y -46.907,Z -112.120,A -90.000,B 90.000,C 0.000} C_DIS
LIN {X 19.737,Y -46.913,Z -112.153,A -90.000,B 90.000,C 0.000} C_DIS
LIN {X 19.859,Y -46.915,Z -112.172,A -90.000,B 90.000,C 0.000} C_DIS
LIN {X 21.230,Y -46.949,Z -112.413,A -90.000,B 90.000,C 0.000} C_DIS
LIN {X 22.662,Y -46.985,Z -112.665,A -90.000,B 90.000,C 0.000} C_DIS
LIN {X 23.033,Y -46.986,Z -112.731,A -90.000,B 90.000,C 0.000} C_DIS
LIN {X 23.887,Y -46.991,Z -112.903,A -90.000,B 90.000,C 0.000} C_DIS
LIN {X 24.081,Y -46.993,Z -112.950,A -90.000,B 90.000,C 0.000} C_DIS
LIN {X 24.400,Y -46.995,Z -113.039,A -90.000,B 90.000,C 0.000} C_DIS
LIN {X 24.594,Y -46.997,Z -113.101,A -90.000,B 90.000,C 0.000} C_DIS
LIN {X 24.693,Y -46.998,Z -113.134,A -90.000,B 90.000,C 0.000} C_DIS
LIN {X 24.838,Y -47.001,Z -113.189,A -90.000,B 90.000,C 0.000} C_DIS
LIN {X 24.998,Y -47.003,Z -113.259,A -90.000,B 90.000,C 0.000} C_DIS
LIN {X 25.388,Y -47.011,Z -113.439,A -90.000,B 90.000,C 0.000} C_DIS
LIN {X 25.525,Y -47.013,Z -113.512,A -90.000,B 90.000,C 0.000} C_DIS
LIN {X 25.656,Y -47.016,Z -113.585,A -90.000,B 90.000,C 0.000} C_DIS
LIN {X 25.796,Y -47.020,Z -113.670,A -90.000,B 90.000,C 0.000} C_DIS
LIN {X 25.952,Y -47.023,Z -113.768,A -90.000,B 90.000,C 0.000} C_DIS
LIN {X 26.100,Y -47.027,Z -113.869,A -90.000,B 90.000,C 0.000} C_DIS
LIN {X 26.266,Y -47.027,Z -113.989,A -90.000,B 90.000,C 0.000} C_DIS
LIN {X 27.535,Y -47.013,Z -114.978,A -90.000,B 90.000,C 0.000} C_DIS
LIN {X 27.805,Y -47.011,Z -115.189,A -90.000,B 90.000,C 0.000} C_DIS
LIN {X 28.279,Y -47.008,Z -115.560,A -90.000,B 90.000,C 0.000} C_DIS
LIN {X 28.471,Y -47.007,Z -115.723,A -90.000,B 90.000,C 0.000} C_DIS
LIN {X 28.631,Y -47.007,Z -115.866,A -90.000,B 90.000,C 0.000} C_DIS
LIN {X 28.758,Y -47.006,Z -115.986,A -90.000,B 90.000,C 0.000} C_DIS
LIN {X 28.917,Y -47.006,Z -116.147,A -90.000,B 90.000,C 0.000} C_DIS
LIN {X 29.063,Y -47.005,Z -116.307,A -90.000,B 90.000,C 0.000} C_DIS
LIN {X 29.809,Y -46.957,Z -117.157,A -90.000,B 90.000,C 0.000} C_DIS
LIN {X 29.940,Y -46.949,Z -117.314,A -90.000,B 90.000,C 0.000} C_DIS
LIN {X 30.164,Y -46.935,Z -117.608,A -90.000,B 90.000,C 0.000} C_DIS
LIN {X 30.287,Y -46.928,Z -117.785,A -90.000,B 90.000,C 0.000} C_DIS
LIN {X 30.431,Y -46.921,Z -118.016,A -90.000,B 90.000,C 0.000} C_DIS
LIN {X 30.528,Y -46.916,Z -118.183,A -90.000,B 90.000,C 0.000} C_DIS
LIN {X 30.682,Y -46.909,Z -118.478,A -90.000,B 90.000,C 0.000} C_DIS
LIN {X 30.761,Y -46.905,Z -118.647,A -90.000,B 90.000,C 0.000} C_DIS
LIN {X 30.855,Y -46.899,Z -118.875,A -90.000,B 90.000,C 0.000} C_DIS
LIN {X 30.908,Y -46.895,Z -119.018,A -90.000,B 90.000,C 0.000} C_DIS
LIN {X 30.992,Y -46.889,Z -119.258,A -90.000,B 90.000,C 0.000} C_DIS
LIN {X 31.052,Y -46.884,Z -119.451,A -90.000,B 90.000,C 0.000} C_DIS
LIN {X 31.110,Y -46.876,Z -119.664,A -90.000,B 90.000,C 0.000} C_DIS
LIN {X 31.189,Y -46.864,Z -120.007,A -90.000,B 90.000,C 0.000} C_DIS
LIN {X 31.214,Y -46.856,Z -120.141,A -90.000,B 90.000,C 0.000} C_DIS
LIN {X 31.400,Y -46.791,Z -121.228,A -90.000,B 90.000,C 0.000} C_DIS
LIN {X 31.446,Y -46.769,Z -121.508,A -90.000,B 90.000,C 0.000} C_DIS
LIN {X 31.458,Y -46.762,Z -121.601,A -90.000,B 90.000,C 0.000} C_DIS
LIN {X 31.473,Y -46.752,Z -121.731,A -90.000,B 90.000,C 0.000} C_DIS
LIN {X 31.489,Y -46.740,Z -121.901,A -90.000,B 90.000,C 0.000} C_DIS
LIN {X 31.503,Y -46.723,Z -122.165,A -90.000,B 90.000,C 0.000} C_DIS
LIN {X 31.507,Y -46.708,Z -122.400,A -90.000,B 90.000,C 0.000} C_DIS
LIN {X 31.498,Y -46.696,Z -122.672,A -90.000,B 90.000,C 0.000} C_DIS
LIN {X 31.482,Y -46.687,Z -122.912,A -90.000,B 90.000,C 0.000} C_DIS
LIN {X 31.453,Y -46.678,Z -123.175,A -90.000,B 90.000,C 0.000} C_DIS
LIN {X 31.433,Y -46.672,Z -123.357,A -90.000,B 90.000,C 0.000} C_DIS
LIN {X 31.439,Y -46.668,Z -123.433,A -90.000,B 90.000,C 0.000} C_DIS
LIN {X 31.511,Y -46.578,Z -124.421,A -90.000,B 90.000,C 0.000} C_DIS
LIN {X 31.516,Y -46.561,Z -124.575,A -90.000,B 90.000,C 0.000} C_DIS
LIN {X 31.513,Y -46.540,Z -124.794,A -90.000,B 90.000,C 0.000} C_DIS
LIN {X 31.502,Y -46.511,Z -125.093,A -90.000,B 90.000,C 0.000} C_DIS
LIN {X 31.497,Y -46.504,Z -125.165,A -90.000,B 90.000,C 0.000} C_DIS
LIN {X 31.474,Y -46.475,Z -125.406,A -90.000,B 90.000,C 0.000} C_DIS
LIN {X 31.428,Y -46.440,Z -125.715,A -90.000,B 90.000,C 0.000} C_DIS
LIN {X 31.383,Y -46.412,Z -125.976,A -90.000,B 90.000,C 0.000} C_DIS
LIN {X 31.350,Y -46.393,Z -126.127,A -90.000,B 90.000,C 0.000} C_DIS
LIN {X 31.206,Y -46.314,Z -126.711,A -90.000,B 90.000,C 0.000} C_DIS
LIN {X 30.867,Y -46.153,Z -128.105,A -90.000,B 90.000,C 0.000} C_DIS
LIN {X 30.805,Y -46.120,Z -128.353,A -90.000,B 90.000,C 0.000} C_DIS
LIN {X 30.736,Y -46.088,Z -128.602,A -90.000,B 90.000,C 0.000} C_DIS
LIN {X 30.706,Y -46.077,Z -128.696,A -90.000,B 90.000,C 0.000} C_DIS
LIN {X 30.599,Y -46.030,Z -129.013,A -90.000,B 90.000,C 0.000} C_DIS
LIN {X 30.472,Y -45.988,Z -129.334,A -90.000,B 90.000,C 0.000} C_DIS
LIN {X 30.377,Y -45.961,Z -129.555,A -90.000,B 90.000,C 0.000} C_DIS
LIN {X 30.285,Y -45.939,Z -129.747,A -90.000,B 90.000,C 0.000} C_DIS
LIN {X 29.323,Y -45.751,Z -131.596,A -90.000,B 90.000,C 0.000} C_DIS
LIN {X 28.983,Y -45.668,Z -132.233,A -90.000,B 90.000,C 0.000} C_DIS
LIN {X 28.623,Y -45.591,Z -132.875,A -90.000,B 90.000,C 0.000} C_DIS
LIN {X 28.495,Y -45.564,Z -133.083,A -90.000,B 90.000,C 0.000} C_DIS
LIN {X 28.363,Y -45.541,Z -133.281,A -90.000,B 90.000,C 0.000} C_DIS
LIN {X 28.301,Y -45.531,Z -133.370,A -90.000,B 90.000,C 0.000} C_DIS
LIN {X 28.114,Y -45.509,Z -133.621,A -90.000,B 90.000,C 0.000} C_DIS
LIN {X 27.993,Y -45.489,Z -133.779,A -90.000,B 90.000,C 0.000} C_DIS
LIN {X 27.360,Y -45.378,Z -134.652,A -90.000,B 90.000,C 0.000} C_DIS
LIN {X 26.989,Y -45.308,Z -135.159,A -90.000,B 90.000,C 0.000} C_DIS
LIN {X 26.989,Y -60.000,Z -135.159,A -90.000,B 90.000,C 0.000} C_DIS
LIN {X -8.367,Y -60.000,Z -137.975,A -90.000,B 90.000,C 0.000} C_DIS
LIN {X -8.367,Y -45.308,Z -137.975,A -90.000,B 90.000,C 0.000} C_DIS
LIN {X -8.561,Y -45.343,Z -137.634,A -90.000,B 90.000,C 0.000} C_DIS
LIN {X -8.666,Y -45.355,Z -137.445,A -90.000,B 90.000,C 0.000} C_DIS
LIN {X -8.822,Y -45.365,Z -137.152,A -90.000,B 90.000,C 0.000} C_DIS
LIN {X -8.903,Y -45.371,Z -136.994,A -90.000,B 90.000,C 0.000} C_DIS
LIN {X -9.021,Y -45.380,Z -136.742,A -90.000,B 90.000,C 0.000} C_DIS
LIN {X -9.103,Y -45.388,Z -136.554,A -90.000,B 90.000,C 0.000} C_DIS
LIN {X -9.188,Y -45.398,Z -136.342,A -90.000,B 90.000,C 0.000} C_DIS
LIN {X -9.458,Y -45.436,Z -135.622,A -90.000,B 90.000,C 0.000} C_DIS
LIN {X -9.519,Y -45.447,Z -135.440,A -90.000,B 90.000,C 0.000} C_DIS
LIN {X -9.570,Y -45.458,Z -135.283,A -90.000,B 90.000,C 0.000} C_DIS
LIN {X -9.611,Y -45.463,Z -135.132,A -90.000,B 90.000,C 0.000} C_DIS
LIN {X -9.718,Y -45.475,Z -134.713,A -90.000,B 90.000,C 0.000} C_DIS
LIN {X -9.762,Y -45.482,Z -134.514,A -90.000,B 90.000,C 0.000} C_DIS
LIN {X -9.815,Y -45.494,Z -134.248,A -90.000,B 90.000,C 0.000} C_DIS
LIN {X -9.860,Y -45.509,Z -133.930,A -90.000,B 90.000,C 0.000} C_DIS
LIN {X -9.888,Y -45.515,Z -133.641,A -90.000,B 90.000,C 0.000} C_DIS
LIN {X -9.919,Y -45.530,Z -133.158,A -90.000,B 90.000,C 0.000} C_DIS
LIN {X -9.923,Y -45.537,Z -132.973,A -90.000,B 90.000,C 0.000} C_DIS
LIN {X -9.922,Y -45.545,Z -132.774,A -90.000,B 90.000,C 0.000} C_DIS
LIN {X -9.916,Y -45.548,Z -132.469,A -90.000,B 90.000,C 0.000} C_DIS
LIN {X -9.902,Y -45.553,Z -132.232,A -90.000,B 90.000,C 0.000} C_DIS
LIN {X -9.866,Y -45.565,Z -131.767,A -90.000,B 90.000,C 0.000} C_DIS
LIN {X -9.730,Y -45.565,Z -130.091,A -90.000,B 90.000,C 0.000} C_DIS
LIN {X -9.695,Y -45.562,Z -129.648,A -90.000,B 90.000,C 0.000} C_DIS
LIN {X -9.685,Y -45.562,Z -129.557,A -90.000,B 90.000,C 0.000} C_DIS
LIN {X -9.654,Y -45.558,Z -129.298,A -90.000,B 90.000,C 0.000} C_DIS
LIN {X -9.630,Y -45.556,Z -129.138,A -90.000,B 90.000,C 0.000} C_DIS
LIN {X -9.590,Y -45.547,Z -128.892,A -90.000,B 90.000,C 0.000} C_DIS
LIN {X -9.423,Y -45.522,Z -128.091,A -90.000,B 90.000,C 0.000} C_DIS
LIN {X -9.368,Y -45.515,Z -127.841,A -90.000,B 90.000,C 0.000} C_DIS
LIN {X -9.300,Y -45.509,Z -127.562,A -90.000,B 90.000,C 0.000} C_DIS
LIN {X -9.235,Y -45.506,Z -127.331,A -90.000,B 90.000,C 0.000} C_DIS
LIN {X -9.137,Y -45.509,Z -127.012,A -90.000,B 90.000,C 0.000} C_DIS
LIN {X -9.074,Y -45.511,Z -126.819,A -90.000,B 90.000,C 0.000} C_DIS
LIN {X -8.987,Y -45.517,Z -126.579,A -90.000,B 90.000,C 0.000} C_DIS
LIN {X -8.920,Y -45.522,Z -126.412,A -90.000,B 90.000,C 0.000} C_DIS
LIN {X -8.829,Y -45.530,Z -126.192,A -90.000,B 90.000,C 0.000} C_DIS
LIN {X -8.712,Y -45.542,Z -125.939,A -90.000,B 90.000,C 0.000} C_DIS
LIN {X -8.598,Y -45.553,Z -125.710,A -90.000,B 90.000,C 0.000} C_DIS
LIN {X -8.396,Y -45.558,Z -125.340,A -90.000,B 90.000,C 0.000} C_DIS
LIN {X -8.146,Y -45.567,Z -124.903,A -90.000,B 90.000,C 0.000} C_DIS
LIN {X -8.057,Y -45.573,Z -124.754,A -90.000,B 90.000,C 0.000} C_DIS
LIN {X -6.926,Y -45.689,Z -122.937,A -90.000,B 90.000,C 0.000} C_DIS
LIN {X -6.629,Y -45.695,Z -122.471,A -90.000,B 90.000,C 0.000} C_DIS
LIN {X -6.409,Y -45.697,Z -122.127,A -90.000,B 90.000,C 0.000} C_DIS
LIN {X -6.230,Y -45.711,Z -121.849,A -90.000,B 90.000,C 0.000} C_DIS
LIN {X -6.139,Y -45.718,Z -121.717,A -90.000,B 90.000,C 0.000} C_DIS
LIN {X -5.868,Y -45.743,Z -121.351,A -90.000,B 90.000,C 0.000} C_DIS
LIN {X -5.443,Y -45.784,Z -120.818,A -90.000,B 90.000,C 0.000} C_DIS
LIN {X -5.328,Y -45.795,Z -120.682,A -90.000,B 90.000,C 0.000} C_DIS
LIN {X -5.091,Y -45.820,Z -120.415,A -90.000,B 90.000,C 0.000} C_DIS
LIN {X -4.859,Y -45.844,Z -120.172,A -90.000,B 90.000,C 0.000} C_DIS
LIN {X -4.751,Y -45.852,Z -120.064,A -90.000,B 90.000,C 0.000} C_DIS
LIN {X -4.058,Y -45.889,Z -119.393,A -90.000,B 90.000,C 0.000} C_DIS
LIN {X -3.056,Y -45.977,Z -118.418,A -90.000,B 90.000,C 0.000} C_DIS
LIN {X -2.258,Y -46.048,Z -117.672,A -90.000,B 90.000,C 0.000} C_DIS
LIN {X -2.097,Y -46.060,Z -117.532,A -90.000,B 90.000,C 0.000} C_DIS
LIN {X -1.862,Y -46.073,Z -117.337,A -90.000,B 90.000,C 0.000} C_DIS
LIN {X -1.688,Y -46.083,Z -117.202,A -90.000,B 90.000,C 0.000} C_DIS
LIN {X -1.252,Y -46.109,Z -116.880,A -90.000,B 90.000,C 0.000} C_DIS
LIN {X 0.699,Y -46.230,Z -115.518,A -90.000,B 90.000,C 0.000} C_DIS
LIN {X 1.087,Y -46.255,Z -115.250,A -90.000,B 90.000,C 0.000} C_DIS
LIN {X 1.264,Y -46.265,Z -115.136,A -90.000,B 90.000,C 0.000} C_DIS
LIN {X 1.387,Y -46.271,Z -115.059,A -90.000,B 90.000,C 0.000} C_DIS
LIN {X 1.695,Y -46.283,Z -114.878,A -90.000,B 90.000,C 0.000} C_DIS
LIN {X 1.802,Y -46.288,Z -114.817,A -90.000,B 90.000,C 0.000} C_DIS
LIN {X 2.007,Y -46.298,Z -114.707,A -90.000,B 90.000,C 0.000} C_DIS
LIN {X 4.243,Y -46.385,Z -113.565,A -90.000,B 90.000,C 0.000} C_DIS
LIN {X 5.438,Y -46.431,Z -112.956,A -90.000,B 90.000,C 0.000} C_DIS
LIN {X 5.740,Y -46.443,Z -112.815,A -90.000,B 90.000,C 0.000} C_DIS
LIN {X 5.885,Y -46.448,Z -112.753,A -90.000,B 90.000,C 0.000} C_DIS
LIN {X 6.317,Y -46.463,Z -112.580,A -90.000,B 90.000,C 0.000} C_DIS
LIN {X 6.565,Y -46.472,Z -112.492,A -90.000,B 90.000,C 0.000} C_DIS
LIN {X 7.152,Y -46.494,Z -112.307,A -90.000,B 90.000,C 0.000} C_DIS
LIN {X 7.502,Y -46.506,Z -112.198,A -90.000,B 90.000,C 0.000} C_DIS
LIN {X 11.458,Y -46.604,Z -110.969,A -90.000,B 90.000,C 0.000} C_DIS
LIN {X 11.779,Y -46.613,Z -110.873,A -90.000,B 90.000,C 0.000} C_DIS
LIN {X 12.092,Y -46.623,Z -110.792,A -90.000,B 90.000,C 0.000} C_DIS
LIN {X 12.234,Y -46.628,Z -110.758,A -90.000,B 90.000,C 0.000} C_DIS
LIN {X 12.492,Y -46.635,Z -110.702,A -90.000,B 90.000,C 0.000} C_DIS
LIN {X 12.867,Y -46.645,Z -110.634,A -90.000,B 90.000,C 0.000} C_DIS
LIN {X 13.105,Y -46.652,Z -110.599,A -90.000,B 90.000,C 0.000} C_DIS
LIN {X 13.384,Y -46.662,Z -110.570,A -90.000,B 90.000,C 0.000} C_DIS
LIN {X 13.701,Y -46.673,Z -110.538,A -90.000,B 90.000,C 0.000} C_DIS
LIN {X 16.442,Y -46.765,Z -110.244,A -90.000,B 90.000,C 0.000} C_DIS
LIN {X 17.539,Y -46.790,Z -110.128,A -90.000,B 90.000,C 0.000} C_DIS
LIN {X 17.885,Y -46.798,Z -110.098,A -90.000,B 90.000,C 0.000} C_DIS
LIN {X 18.157,Y -46.805,Z -110.086,A -90.000,B 90.000,C 0.000} C_DIS
LIN {X 18.308,Y -46.809,Z -110.081,A -90.000,B 90.000,C 0.000} C_DIS
LIN {X 18.909,Y -46.825,Z -110.080,A -90.000,B 90.000,C 0.000} C_DIS
LIN {X 19.128,Y -46.831,Z -110.088,A -90.000,B 90.000,C 0.000} C_DIS
LIN {X 19.608,Y -46.844,Z -110.126,A -90.000,B 90.000,C 0.000} C_DIS
LIN {X 19.751,Y -46.848,Z -110.142,A -90.000,B 90.000,C 0.000} C_DIS
LIN {X 19.951,Y -46.854,Z -110.165,A -90.000,B 90.000,C 0.000} C_DIS
LIN {X 20.205,Y -46.863,Z -110.203,A -90.000,B 90.000,C 0.000} C_DIS
LIN {X 21.007,Y -46.881,Z -110.344,A -90.000,B 90.000,C 0.000} C_DIS
LIN {X 23.429,Y -46.950,Z -110.771,A -90.000,B 90.000,C 0.000} C_DIS
LIN {X 24.017,Y -46.965,Z -110.889,A -90.000,B 90.000,C 0.000} C_DIS
LIN {X 24.357,Y -46.966,Z -110.959,A -90.000,B 90.000,C 0.000} C_DIS
LIN {X 24.619,Y -46.966,Z -111.024,A -90.000,B 90.000,C 0.000} C_DIS
LIN {X 24.997,Y -46.968,Z -111.130,A -90.000,B 90.000,C 0.000} C_DIS
LIN {X 25.329,Y -46.972,Z -111.239,A -90.000,B 90.000,C 0.000} C_DIS
LIN {X 25.549,Y -46.974,Z -111.320,A -90.000,B 90.000,C 0.000} C_DIS
LIN {X 25.632,Y -46.975,Z -111.354,A -90.000,B 90.000,C 0.000} C_DIS
LIN {X 25.951,Y -46.978,Z -111.496,A -90.000,B 90.000,C 0.000} C_DIS
LIN {X 26.229,Y -46.981,Z -111.625,A -90.000,B 90.000,C 0.000} C_DIS
LIN {X 26.394,Y -46.982,Z -111.709,A -90.000,B 90.000,C 0.000} C_DIS
LIN {X 26.567,Y -46.984,Z -111.803,A -90.000,B 90.000,C 0.000} C_DIS
LIN {X 26.693,Y -46.985,Z -111.875,A -90.000,B 90.000,C 0.000} C_DIS
LIN {X 26.861,Y -46.986,Z -111.977,A -90.000,B 90.000,C 0.000} C_DIS
LIN {X 27.078,Y -46.988,Z -112.115,A -90.000,B 90.000,C 0.000} C_DIS
LIN {X 27.291,Y -46.990,Z -112.262,A -90.000,B 90.000,C 0.000} C_DIS
LIN {X 27.426,Y -46.988,Z -112.361,A -90.000,B 90.000,C 0.000} C_DIS
LIN {X 27.717,Y -46.975,Z -112.585,A -90.000,B 90.000,C 0.000} C_DIS
LIN {X 28.361,Y -46.963,Z -113.087,A -90.000,B 90.000,C 0.000} C_DIS
LIN {X 29.512,Y -46.949,Z -113.987,A -90.000,B 90.000,C 0.000} C_DIS
LIN {X 29.766,Y -46.946,Z -114.200,A -90.000,B 90.000,C 0.000} C_DIS
LIN {X 29.995,Y -46.945,Z -114.405,A -90.000,B 90.000,C 0.000} C_DIS
LIN {X 30.118,Y -46.945,Z -114.521,A -90.000,B 90.000,C 0.000} C_DIS
LIN {X 30.262,Y -46.943,Z -114.664,A -90.000,B 90.000,C 0.000} C_DIS
LIN {X 30.392,Y -46.934,Z -114.798,A -90.000,B 90.000,C 0.000} C_DIS
LIN {X 30.568,Y -46.923,Z -114.992,A -90.000,B 90.000,C 0.000} C_DIS
LIN {X 31.347,Y -46.871,Z -115.881,A -90.000,B 90.000,C 0.000} C_DIS
LIN {X 31.538,Y -46.858,Z -116.115,A -90.000,B 90.000,C 0.000} C_DIS
LIN {X 31.759,Y -46.843,Z -116.404,A -90.000,B 90.000,C 0.000} C_DIS
LIN {X 31.904,Y -46.834,Z -116.611,A -90.000,B 90.000,C 0.000} C_DIS
LIN {X 31.981,Y -46.829,Z -116.726,A -90.000,B 90.000,C 0.000} C_DIS
LIN {X 32.158,Y -46.818,Z -117.012,A -90.000,B 90.000,C 0.000} C_DIS
LIN {X 32.246,Y -46.812,Z -117.165,A -90.000,B 90.000,C 0.000} C_DIS
LIN {X 32.299,Y -46.808,Z -117.259,A -90.000,B 90.000,C 0.000} C_DIS
LIN {X 32.479,Y -46.797,Z -117.609,A -90.000,B 90.000,C 0.000} C_DIS
LIN {X 32.605,Y -46.781,Z -117.883,A -90.000,B 90.000,C 0.000} C_DIS
LIN {X 32.708,Y -46.766,Z -118.134,A -90.000,B 90.000,C 0.000} C_DIS
LIN {X 32.800,Y -46.745,Z -118.387,A -90.000,B 90.000,C 0.000} C_DIS
LIN {X 32.867,Y -46.730,Z -118.580,A -90.000,B 90.000,C 0.000} C_DIS
LIN {X 32.962,Y -46.705,Z -118.885,A -90.000,B 90.000,C 0.000} C_DIS
LIN {X 33.032,Y -46.686,Z -119.144,A -90.000,B 90.000,C 0.000} C_DIS
LIN {X 33.138,Y -46.655,Z -119.609,A -90.000,B 90.000,C 0.000} C_DIS
LIN {X 33.189,Y -46.638,Z -119.891,A -90.000,B 90.000,C 0.000} C_DIS
LIN {X 33.337,Y -46.587,Z -120.755,A -90.000,B 90.000,C 0.000} C_DIS
LIN {X 33.360,Y -46.576,Z -120.890,A -90.000,B 90.000,C 0.000} C_DIS
LIN {X 33.413,Y -46.550,Z -121.221,A -90.000,B 90.000,C 0.000} C_DIS
LIN {X 33.442,Y -46.533,Z -121.452,A -90.000,B 90.000,C 0.000} C_DIS
LIN {X 33.470,Y -46.512,Z -121.746,A -90.000,B 90.000,C 0.000} C_DIS
LIN {X 33.489,Y -46.487,Z -122.121,A -90.000,B 90.000,C 0.000} C_DIS
LIN {X 33.490,Y -46.480,Z -122.227,A -90.000,B 90.000,C 0.000} C_DIS
LIN {X 33.492,Y -46.468,Z -122.356,A -90.000,B 90.000,C 0.000} C_DIS
LIN {X 33.490,Y -46.459,Z -122.452,A -90.000,B 90.000,C 0.000} C_DIS
LIN {X 33.476,Y -46.428,Z -122.795,A -90.000,B 90.000,C 0.000} C_DIS
LIN {X 33.459,Y -46.409,Z -123.022,A -90.000,B 90.000,C 0.000} C_DIS
LIN {X 33.445,Y -46.395,Z -123.158,A -90.000,B 90.000,C 0.000} C_DIS
LIN {X 33.419,Y -46.373,Z -123.378,A -90.000,B 90.000,C 0.000} C_DIS
LIN {X 33.475,Y -46.235,Z -124.261,A -90.000,B 90.000,C 0.000} C_DIS
LIN {X 33.482,Y -46.197,Z -124.512,A -90.000,B 90.000,C 0.000} C_DIS
LIN {X 33.473,Y -46.149,Z -124.868,A -90.000,B 90.000,C 0.000} C_DIS
LIN {X 33.461,Y -46.109,Z -125.161,A -90.000,B 90.000,C 0.000} C_DIS
LIN {X 33.435,Y -46.074,Z -125.447,A -90.000,B 90.000,C 0.000} C_DIS
LIN {X 33.420,Y -46.051,Z -125.594,A -90.000,B 90.000,C 0.000} C_DIS
LIN {X 33.355,Y -45.989,Z -126.002,A -90.000,B 90.000,C 0.000} C_DIS
LIN {X 33.294,Y -45.941,Z -126.327,A -90.000,B 90.000,C 0.000} C_DIS
LIN {X 33.249,Y -45.913,Z -126.529,A -90.000,B 90.000,C 0.000} C_DIS
LIN {X 33.052,Y -45.805,Z -127.329,A -90.000,B 90.000,C 0.000} C_DIS
LIN {X 32.843,Y -45.687,Z -128.164,A -90.000,B 90.000,C 0.000} C_DIS
LIN {X 32.831,Y -45.679,Z -128.210,A -90.000,B 90.000,C 0.000} C_DIS
LIN {X 32.671,Y -45.557,Z -128.802,A -90.000,B 90.000,C 0.000} C_DIS
LIN {X 32.574,Y -45.495,Z -129.121,A -90.000,B 90.000,C 0.000} C_DIS
LIN {X 32.430,Y -45.418,Z -129.537,A -90.000,B 90.000,C 0.000} C_DIS
LIN {X 32.413,Y -45.410,Z -129.584,A -90.000,B 90.000,C 0.000} C_DIS
LIN {X 32.236,Y -45.339,Z -130.016,A -90.000,B 90.000,C 0.000} C_DIS
LIN {X 32.150,Y -45.308,Z -130.211,A -90.000,B 90.000,C 0.000} C_DIS
LIN {X 32.150,Y -60.000,Z -130.211,A -90.000,B 90.000,C 0.000} C_DIS
LIN {X -8.019,Y -60.000,Z -121.005,A -90.000,B 90.000,C 0.000} C_DIS
LIN {X -8.019,Y -45.308,Z -121.005,A -90.000,B 90.000,C 0.000} C_DIS
LIN {X -7.834,Y -45.323,Z -120.718,A -90.000,B 90.000,C 0.000} C_DIS
LIN {X -7.661,Y -45.338,Z -120.474,A -90.000,B 90.000,C 0.000} C_DIS
LIN {X -7.575,Y -45.346,Z -120.359,A -90.000,B 90.000,C 0.000} C_DIS
LIN {X -7.391,Y -45.373,Z -120.109,A -90.000,B 90.000,C 0.000} C_DIS
LIN {X -6.938,Y -45.441,Z -119.535,A -90.000,B 90.000,C 0.000} C_DIS
LIN {X -6.787,Y -45.463,Z -119.354,A -90.000,B 90.000,C 0.000} C_DIS
LIN {X -6.699,Y -45.475,Z -119.254,A -90.000,B 90.000,C 0.000} C_DIS
LIN {X -6.501,Y -45.493,Z -119.034,A -90.000,B 90.000,C 0.000} C_DIS
LIN {X -6.241,Y -45.517,Z -118.764,A -90.000,B 90.000,C 0.000} C_DIS
LIN {X -6.115,Y -45.530,Z -118.637,A -90.000,B 90.000,C 0.000} C_DIS
LIN {X -4.925,Y -45.648,Z -117.475,A -90.000,B 90.000,C 0.000} C_DIS
LIN {X -4.398,Y -45.719,Z -116.957,A -90.000,B 90.000,C 0.000} C_DIS
LIN {X -4.198,Y -45.743,Z -116.769,A -90.000,B 90.000,C 0.000} C_DIS
LIN {X -3.551,Y -45.800,Z -116.166,A -90.000,B 90.000,C 0.000} C_DIS
LIN {X -3.354,Y -45.818,Z -115.995,A -90.000,B 90.000,C 0.000} C_DIS
LIN {X -3.074,Y -45.844,Z -115.763,A -90.000,B 90.000,C 0.000} C_DIS
LIN {X -2.861,Y -45.864,Z -115.597,A -90.000,B 90.000,C 0.000} C_DIS
LIN {X -2.609,Y -45.888,Z -115.410,A -90.000,B 90.000,C 0.000} C_DIS
LIN {X -2.382,Y -45.905,Z -115.242,A -90.000,B 90.000,C 0.000} C_DIS
LIN {X -0.938,Y -46.019,Z -114.231,A -90.000,B 90.000,C 0.000} C_DIS
LIN {X -0.038,Y -46.065,Z -113.607,A -90.000,B 90.000,C 0.000} C_DIS
LIN {X 0.309,Y -46.084,Z -113.384,A -90.000,B 90.000,C 0.000} C_DIS
LIN {X 0.384,Y -46.088,Z -113.338,A -90.000,B 90.000,C 0.000} C_DIS
LIN {X 0.718,Y -46.108,Z -113.142,A -90.000,B 90.000,C 0.000} C_DIS
LIN {X 0.867,Y -46.118,Z -113.058,A -90.000,B 90.000,C 0.000} C_DIS
LIN {X 1.106,Y -46.134,Z -112.929,A -90.000,B 90.000,C 0.000} C_DIS
LIN {X 2.993,Y -46.260,Z -111.961,A -90.000,B 90.000,C 0.000} C_DIS
LIN {X 4.382,Y -46.330,Z -111.252,A -90.000,B 90.000,C 0.000} C_DIS
LIN {X 4.595,Y -46.338,Z -111.145,A -90.000,B 90.000,C 0.000} C_DIS
LIN {X 4.956,Y -46.350,Z -110.978,A -90.000,B 90.000,C 0.000} C_DIS
LIN {X 5.160,Y -46.357,Z -110.891,A -90.000,B 90.000,C 0.000} C_DIS
LIN {X 5.649,Y -46.373,Z -110.697,A -90.000,B 90.000,C 0.000} C_DIS
LIN {X 5.969,Y -46.384,Z -110.585,A -90.000,B 90.000,C 0.000} C_DIS
LIN {X 7.894,Y -46.450,Z -109.983,A -90.000,B 90.000,C 0.000} C_DIS
LIN {X 9.399,Y -46.504,Z -109.515,A -90.000,B 90.000,C 0.000} C_DIS
LIN {X 10.890,Y -46.550,Z -109.052,A -90.000,B 90.000,C 0.000} C_DIS
LIN {X 11.278,Y -46.562,Z -108.938,A -90.000,B 90.000,C 0.000} C_DIS
LIN {X 11.689,Y -46.575,Z -108.832,A -90.000,B 90.000,C 0.000} C_DIS
LIN {X 11.817,Y -46.579,Z -108.802,A -90.000,B 90.000,C 0.000} C_DIS
LIN {X 12.134,Y -46.589,Z -108.735,A -90.000,B 90.000,C 0.000} C_DIS
LIN {X 12.620,Y -46.604,Z -108.649,A -90.000,B 90.000,C 0.000} C_DIS
LIN {X 12.822,Y -46.610,Z -108.620,A -90.000,B 90.000,C 0.000} C_DIS
LIN {X 13.340,Y -46.625,Z -108.565,A -90.000,B 90.000,C 0.000} C_DIS
LIN {X 13.973,Y -46.647,Z -108.498,A -90.000,B 90.000,C 0.000} C_DIS
LIN {X 14.110,Y -46.651,Z -108.483,A -90.000,B 90.000,C 0.000} C_DIS
LIN {X 17.368,Y -46.810,Z -108.135,A -90.000,B 90.000,C 0.000} C_DIS
LIN {X 17.714,Y -46.826,Z -108.105,A -90.000,B 90.000,C 0.000} C_DIS
LIN {X 18.026,Y -46.840,Z -108.090,A -90.000,B 90.000,C 0.000} C_DIS
LIN {X 18.327,Y -46.852,Z -108.082,A -90.000,B 90.000,C 0.000} C_DIS
LIN {X 18.904,Y -46.874,Z -108.081,A -90.000,B 90.000,C 0.000} C_DIS
LIN {X 19.148,Y -46.883,Z -108.089,A -90.000,B 90.000,C 0.000} C_DIS
LIN {X 19.275,Y -46.887,Z -108.094,A -90.000,B 90.000,C 0.000} C_DIS
LIN {X 19.815,Y -46.906,Z -108.138,A -90.000,B 90.000,C 0.000} C_DIS
LIN {X 20.186,Y -46.918,Z -108.180,A -90.000,B 90.000,C 0.000} C_DIS
LIN {X 20.550,Y -46.930,Z -108.234,A -90.000,B 90.000,C 0.000} C_DIS
LIN {X 21.362,Y -46.958,Z -108.377,A -90.000,B 90.000,C 0.000} C_DIS
LIN {X 21.700,Y -46.969,Z -108.437,A -90.000,B 90.000,C 0.000} C_DIS
LIN {X 23.774,Y -47.012,Z -108.801,A -90.000,B 90.000,C 0.000} C_DIS
LIN {X 24.600,Y -47.028,Z -108.968,A -90.000,B 90.000,C 0.000} C_DIS
LIN {X 24.851,Y -47.033,Z -109.022,A -90.000,B 90.000,C 0.000} C_DIS
LIN {X 25.160,Y -47.039,Z -109.100,A -90.000,B 90.000,C 0.000} C_DIS
LIN {X 25.538,Y -47.040,Z -109.206,A -90.000,B 90.000,C 0.000} C_DIS
LIN {X 25.781,Y -47.040,Z -109.284,A -90.000,B 90.000,C 0.000} C_DIS
LIN {X 25.976,Y -47.039,Z -109.347,A -90.000,B 90.000,C 0.000} C_DIS
LIN {X 26.247,Y -47.039,Z -109.447,A -90.000,B 90.000,C 0.000} C_DIS
LIN {X 26.425,Y -47.038,Z -109.519,A -90.000,B 90.000,C 0.000} C_DIS
LIN {X 26.869,Y -47.035,Z -109.718,A -90.000,B 90.000,C 0.000} C_DIS
LIN {X 27.135,Y -47.034,Z -109.843,A -90.000,B 90.000,C 0.000} C_DIS
LIN {X 27.348,Y -47.032,Z -109.952,A -90.000,B 90.000,C 0.000} C_DIS
LIN {X 27.557,Y -47.030,Z -110.066,A -90.000,B 90.000,C 0.000} C_DIS
LIN {X 27.758,Y -47.028,Z -110.182,A -90.000,B 90.000,C 0.000} C_DIS
LIN {X 27.936,Y -47.026,Z -110.291,A -90.000,B 90.000,C 0.000} C_DIS
LIN {X 28.116,Y -47.024,Z -110.406,A -90.000,B 90.000,C 0.000} C_DIS
LIN {X 28.222,Y -47.025,Z -110.475,A -90.000,B 90.000,C 0.000} C_DIS
LIN {X 28.471,Y -47.026,Z -110.647,A -90.000,B 90.000,C 0.000} C_DIS
LIN {X 28.650,Y -47.019,Z -110.779,A -90.000,B 90.000,C 0.000} C_DIS
LIN {X 28.715,Y -47.016,Z -110.829,A -90.000,B 90.000,C 0.000} C_DIS
LIN {X 30.149,Y -46.950,Z -111.946,A -90.000,B 90.000,C 0.000} C_DIS
LIN {X 30.262,Y -46.945,Z -112.035,A -90.000,B 90.000,C 0.000} C_DIS
LIN {X 30.798,Y -46.934,Z -112.455,A -90.000,B 90.000,C 0.000} C_DIS
LIN {X 31.102,Y -46.927,Z -112.711,A -90.000,B 90.000,C 0.000} C_DIS
LIN {X 31.389,Y -46.921,Z -112.971,A -90.000,B 90.000,C 0.000} C_DIS
LIN {X 31.565,Y -46.904,Z -113.140,A -90.000,B 90.000,C 0.000} C_DIS
LIN {X 31.748,Y -46.885,Z -113.324,A -90.000,B 90.000,C 0.000} C_DIS
LIN {X 31.871,Y -46.873,Z -113.452,A -90.000,B 90.000,C 0.000} C_DIS
LIN {X 32.070,Y -46.852,Z -113.673,A -90.000,B 90.000,C 0.000} C_DIS
LIN {X 32.170,Y -46.841,Z -113.787,A -90.000,B 90.000,C 0.000} C_DIS
LIN {X 32.848,Y -46.793,Z -114.561,A -90.000,B 90.000,C 0.000} C_DIS
LIN {X 33.085,Y -46.775,Z -114.850,A -90.000,B 90.000,C 0.000} C_DIS
LIN {X 33.344,Y -46.756,Z -115.188,A -90.000,B 90.000,C 0.000} C_DIS
LIN {X 33.510,Y -46.744,Z -115.422,A -90.000,B 90.000,C 0.000} C_DIS
LIN {X 33.642,Y -46.734,Z -115.616,A -90.000,B 90.000,C 0.000} C_DIS
LIN {X 33.796,Y -46.723,Z -115.863,A -90.000,B 90.000,C 0.000} C_DIS
LIN {X 33.878,Y -46.714,Z -115.997,A -90.000,B 90.000,C 0.000} C_DIS
LIN {X 34.025,Y -46.696,Z -116.255,A -90.000,B 90.000,C 0.000} C_DIS
LIN {X 34.103,Y -46.682,Z -116.402,A -90.000,B 90.000,C 0.000} C_DIS
LIN {X 34.289,Y -46.646,Z -116.772,A -90.000,B 90.000,C 0.000} C_DIS
LIN {X 34.446,Y -46.614,Z -117.119,A -90.000,B 90.000,C 0.000} C_DIS
LIN {X 34.571,Y -46.587,Z -117.429,A -90.000,B 90.000,C 0.000} C_DIS
LIN {X 34.649,Y -46.569,Z -117.643,A -90.000,B 90.000,C 0.000} C_DIS
LIN {X 34.763,Y -46.542,Z -117.973,A -90.000,B 90.000,C 0.000} C_DIS
LIN {X 34.881,Y -46.512,Z -118.355,A -90.000,B 90.000,C 0.000} C_DIS
LIN {X 34.970,Y -46.488,Z -118.691,A -90.000,B 90.000,C 0.000} C_DIS
LIN {X 35.082,Y -46.453,Z -119.185,A -90.000,B 90.000,C 0.000} C_DIS
LIN {X 35.147,Y -46.430,Z -119.542,A -90.000,B 90.000,C 0.000} C_DIS
LIN {X 35.253,Y -46.391,Z -120.163,A -90.000,B 90.000,C 0.000} C_DIS
LIN {X 35.339,Y -46.328,Z -120.691,A -90.000,B 90.000,C 0.000} C_DIS
LIN {X 35.368,Y -46.303,Z -120.883,A -90.000,B 90.000,C 0.000} C_DIS
LIN {X 35.406,Y -46.258,Z -121.198,A -90.000,B 90.000,C 0.000} C_DIS
LIN {X 35.436,Y -46.211,Z -121.537,A -90.000,B 90.000,C 0.000} C_DIS
LIN {X 35.442,Y -46.200,Z -121.627,A -90.000,B 90.000,C 0.000} C_DIS
LIN {X 35.458,Y -46.143,Z -122.070,A -90.000,B 90.000,C 0.000} C_DIS
LIN {X 35.459,Y -46.107,Z -122.373,A -90.000,B 90.000,C 0.000} C_DIS
LIN {X 35.456,Y -46.093,Z -122.496,A -90.000,B 90.000,C 0.000} C_DIS
LIN {X 35.440,Y -46.055,Z -122.840,A -90.000,B 90.000,C 0.000} C_DIS
LIN {X 35.417,Y -46.015,Z -123.134,A -90.000,B 90.000,C 0.000} C_DIS
LIN {X 35.390,Y -45.984,Z -123.384,A -90.000,B 90.000,C 0.000} C_DIS
LIN {X 35.436,Y -45.860,Z -124.151,A -90.000,B 90.000,C 0.000} C_DIS
LIN {X 35.443,Y -45.822,Z -124.402,A -90.000,B 90.000,C 0.000} C_DIS
LIN {X 35.442,Y -45.801,Z -124.540,A -90.000,B 90.000,C 0.000} C_DIS
LIN {X 35.433,Y -45.749,Z -124.901,A -90.000,B 90.000,C 0.000} C_DIS
LIN {X 35.419,Y -45.702,Z -125.169,A -90.000,B 90.000,C 0.000} C_DIS
LIN {X 35.410,Y -45.681,Z -125.286,A -90.000,B 90.000,C 0.000} C_DIS
LIN {X 35.373,Y -45.617,Z -125.657,A -90.000,B 90.000,C 0.000} C_DIS
LIN {X 35.350,Y -45.581,Z -125.828,A -90.000,B 90.000,C 0.000} C_DIS
LIN {X 35.268,Y -45.487,Z -126.300,A -90.000,B 90.000,C 0.000} C_DIS
LIN {X 35.193,Y -45.416,Z -126.675,A -90.000,B 90.000,C 0.000} C_DIS
LIN {X 35.146,Y -45.379,Z -126.875,A -90.000,B 90.000,C 0.000} C_DIS
LIN {X 35.042,Y -45.308,Z -127.280,A -90.000,B 90.000,C 0.000} C_DIS
LIN {X 35.004,Y -45.282,Z -127.433,A -90.000,B 90.000,C 0.000} C_DIS
LIN {X 34.972,Y -45.255,Z -127.578,A -90.000,B 90.000,C 0.000} C_DIS
LIN {X 34.946,Y -45.229,Z -127.714,A -90.000,B 90.000,C 0.000} C_DIS
LIN {X 34.908,Y -45.180,Z -127.961,A -90.000,B 90.000,C 0.000} C_DIS
LIN {X 34.897,Y -45.156,Z -128.073,A -90.000,B 90.000,C 0.000} C_DIS
LIN {X 34.891,Y -45.133,Z -128.177,A -90.000,B 90.000,C 0.000} C_DIS
LIN {X 34.889,Y -45.111,Z -128.273,A -90.000,B 90.000,C 0.000} C_DIS
LIN {X 34.895,Y -45.080,Z -128.402,A -90.000,B 90.000,C 0.000} C_DIS
LIN {X 34.904,Y -45.060,Z -128.479,A -90.000,B 90.000,C 0.000} C_DIS
LIN {X 34.926,Y -45.031,Z -128.580,A -90.000,B 90.000,C 0.000} C_DIS
LIN {X 34.945,Y -45.013,Z -128.638,A -90.000,B 90.000,C 0.000} C_DIS
LIN {X 34.981,Y -44.988,Z -128.713,A -90.000,B 90.000,C 0.000} C_DIS
LIN {X 35.009,Y -44.972,Z -128.753,A -90.000,B 90.000,C 0.000} C_DIS
LIN {X 35.058,Y -44.950,Z -128.802,A -90.000,B 90.000,C 0.000} C_DIS
LIN {X 35.113,Y -44.929,Z -128.835,A -90.000,B 90.000,C 0.000} C_DIS
LIN {X 35.175,Y -44.911,Z -128.853,A -90.000,B 90.000,C 0.000} C_DIS
LIN {X 35.220,Y -44.899,Z -128.858,A -90.000,B 90.000,C 0.000} C_DIS
LIN {X 35.291,Y -44.884,Z -128.853,A -90.000,B 90.000,C 0.000} C_DIS
LIN {X 35.368,Y -44.870,Z -128.834,A -90.000,B 90.000,C 0.000} C_DIS
LIN {X 35.449,Y -44.859,Z -128.802,A -90.000,B 90.000,C 0.000} C_DIS
LIN {X 35.505,Y -44.853,Z -128.774,A -90.000,B 90.000,C 0.000} C_DIS
LIN {X 35.592,Y -44.844,Z -128.720,A -90.000,B 90.000,C 0.000} C_DIS
LIN {X 35.713,Y -44.837,Z -128.630,A -90.000,B 90.000,C 0.000} C_DIS
LIN {X 35.775,Y -44.834,Z -128.577,A -90.000,B 90.000,C 0.000} C_DIS
LIN {X 35.902,Y -44.832,Z -128.457,A -90.000,B 90.000,C 0.000} C_DIS
LIN {X 35.966,Y -44.833,Z -128.389,A -90.000,B 90.000,C 0.000} C_DIS
LIN {X 36.096,Y -44.836,Z -128.239,A -90.000,B 90.000,C 0.000} C_DIS
LIN {X 36.226,Y -44.843,Z -128.071,A -90.000,B 90.000,C 0.000} C_DIS
LIN {X 36.291,Y -44.849,Z -127.981,A -90.000,B 90.000,C 0.000} C_DIS
LIN {X 36.419,Y -44.862,Z -127.787,A -90.000,B 90.000,C 0.000} C_DIS
LIN {X 36.545,Y -44.879,Z -127.578,A -90.000,B 90.000,C 0.000} C_DIS
LIN {X 36.606,Y -44.889,Z -127.468,A -90.000,B 90.000,C 0.000} C_DIS
LIN {X 36.725,Y -44.912,Z -127.237,A -90.000,B 90.000,C 0.000} C_DIS
LIN {X 36.839,Y -44.939,Z -126.992,A -90.000,B 90.000,C 0.000} C_DIS
LIN {X 36.945,Y -44.970,Z -126.734,A -90.000,B 90.000,C 0.000} C_DIS
LIN {X 37.043,Y -45.006,Z -126.465,A -90.000,B 90.000,C 0.000} C_DIS
LIN {X 37.088,Y -45.025,Z -126.326,A -90.000,B 90.000,C 0.000} C_DIS
LIN {X 37.171,Y -45.067,Z -126.041,A -90.000,B 90.000,C 0.000} C_DIS
LIN {X 37.242,Y -45.113,Z -125.747,A -90.000,B 90.000,C 0.000} C_DIS
LIN {X 37.300,Y -45.163,Z -125.444,A -90.000,B 90.000,C 0.000} C_DIS
LIN {X 37.324,Y -45.190,Z -125.289,A -90.000,B 90.000,C 0.000} C_DIS
LIN {X 37.353,Y -45.232,Z -125.054,A -90.000,B 90.000,C 0.000} C_DIS
LIN {X 37.373,Y -45.279,Z -124.816,A -90.000,B 90.000,C 0.000} C_DIS
LIN {X 37.382,Y -45.308,Z -124.655,A -90.000,B 90.000,C 0.000} C_DIS
LIN {X 37.384,Y -45.318,Z -124.606,A -90.000,B 90.000,C 0.000} C_DIS
LIN {X 37.390,Y -45.370,Z -124.346,A -90.000,B 90.000,C 0.000} C_DIS
LIN {X 37.387,Y -45.436,Z -124.033,A -90.000,B 90.000,C 0.000} C_DIS
LIN {X 37.366,Y -45.535,Z -123.578,A -90.000,B 90.000,C 0.000} C_DIS
LIN {X 37.356,Y -45.578,Z -123.373,A -90.000,B 90.000,C 0.000} C_DIS
LIN {X 37.365,Y -45.591,Z -123.291,A -90.000,B 90.000,C 0.000} C_DIS
LIN {X 37.394,Y -45.644,Z -122.961,A -90.000,B 90.000,C 0.000} C_DIS
LIN {X 37.408,Y -45.682,Z -122.737,A -90.000,B 90.000,C 0.000} C_DIS
LIN {X 37.417,Y -45.705,Z -122.570,A -90.000,B 90.000,C 0.000} C_DIS
LIN {X 37.424,Y -45.740,Z -122.323,A -90.000,B 90.000,C 0.000} C_DIS
LIN {X 37.424,Y -45.776,Z -122.022,A -90.000,B 90.000,C 0.000} C_DIS
LIN {X 37.406,Y -45.837,Z -121.524,A -90.000,B 90.000,C 0.000} C_DIS
LIN {X 37.397,Y -45.857,Z -121.367,A -90.000,B 90.000,C 0.000} C_DIS
LIN {X 37.363,Y -45.907,Z -120.979,A -90.000,B 90.000,C 0.000} C_DIS
LIN {X 37.318,Y -45.960,Z -120.598,A -90.000,B 90.000,C 0.000} C_DIS
LIN {X 37.272,Y -46.003,Z -120.292,A -90.000,B 90.000,C 0.000} C_DIS
LIN {X 37.096,Y -46.152,Z -119.191,A -90.000,B 90.000,C 0.000} C_DIS
LIN {X 37.029,Y -46.205,Z -118.802,A -90.000,B 90.000,C 0.000} C_DIS
LIN {X 37.008,Y -46.220,Z -118.700,A -90.000,B 90.000,C 0.000} C_DIS
LIN {X 36.907,Y -46.279,Z -118.238,A -90.000,B 90.000,C 0.000} C_DIS
LIN {X 36.860,Y -46.303,Z -118.054,A -90.000,B 90.000,C 0.000} C_DIS
LIN {X 36.802,Y -46.319,Z -117.833,A -90.000,B 90.000,C 0.000} C_DIS
LIN {X 36.742,Y -46.335,Z -117.632,A -90.000,B 90.000,C 0.000} C_DIS
LIN {X 36.638,Y -46.360,Z -117.299,A -90.000,B 90.000,C 0.000} C_DIS
LIN {X 36.514,Y -46.388,Z -116.943,A -90.000,B 90.000,C 0.000} C_DIS
LIN {X 36.445,Y -46.403,Z -116.756,A -90.000,B 90.000,C 0.000} C_DIS
LIN {X 36.365,Y -46.419,Z -116.552,A -90.000,B 90.000,C 0.000} C_DIS
LIN {X 36.257,Y -46.440,Z -116.289,A -90.000,B 90.000,C 0.000} C_DIS
LIN {X 36.100,Y -46.470,Z -115.941,A -90.000,B 90.000,C 0.000} C_DIS
LIN {X 35.878,Y -46.512,Z -115.497,A -90.000,B 90.000,C 0.000} C_DIS
LIN {X 35.782,Y -46.533,Z -115.313,A -90.000,B 90.000,C 0.000} C_DIS
LIN {X 35.576,Y -46.578,Z -114.948,A -90.000,B 90.000,C 0.000} C_DIS
LIN {X 35.334,Y -46.629,Z -114.555,A -90.000,B 90.000,C 0.000} C_DIS
LIN {X 35.254,Y -46.645,Z -114.434,A -90.000,B 90.000,C 0.000} C_DIS
LIN {X 35.160,Y -46.657,Z -114.295,A -90.000,B 90.000,C 0.000} C_DIS
LIN {X 34.945,Y -46.683,Z -113.991,A -90.000,B 90.000,C 0.000} C_DIS
LIN {X 34.668,Y -46.703,Z -113.630,A -90.000,B 90.000,C 0.000} C_DIS
LIN {X 34.391,Y -46.723,Z -113.291,A -90.000,B 90.000,C 0.000} C_DIS
LIN {X 33.573,Y -46.810,Z -112.354,A -90.000,B 90.000,C 0.000} C_DIS
LIN {X 33.308,Y -46.837,Z -112.062,A -90.000,B 90.000,C 0.000} C_DIS
LIN {X 33.190,Y -46.849,Z -111.939,A -90.000,B 90.000,C 0.000} C_DIS
LIN {X 33.004,Y -46.865,Z -111.751,A -90.000,B 90.000,C 0.000} C_DIS
LIN {X 32.787,Y -46.883,Z -111.540,A -90.000,B 90.000,C 0.000} C_DIS
LIN {X 32.447,Y -46.921,Z -111.231,A -90.000,B 90.000,C 0.000} C_DIS
LIN {X 32.087,Y -46.936,Z -110.926,A -90.000,B 90.000,C 0.000} C_DIS
LIN {X 31.874,Y -46.944,Z -110.757,A -90.000,B 90.000,C 0.000} C_DIS
LIN {X 30.658,Y -46.991,Z -109.807,A -90.000,B 90.000,C 0.000} C_DIS
LIN {X 29.834,Y -47.056,Z -109.168,A -90.000,B 90.000,C 0.000} C_DIS
LIN {X 29.684,Y -47.068,Z -109.057,A -90.000,B 90.000,C 0.000} C_DIS
LIN {X 29.531,Y -47.079,Z -108.950,A -90.000,B 90.000,C 0.000} C_DIS
LIN {X 29.324,Y -47.084,Z -108.807,A -90.000,B 90.000,C 0.000} C_DIS
LIN {X 29.021,Y -47.087,Z -108.612,A -90.000,B 90.000,C 0.000} C_DIS
LIN {X 28.847,Y -47.089,Z -108.505,A -90.000,B 90.000,C 0.000} C_DIS
LIN {X 28.560,Y -47.092,Z -108.336,A -90.000,B 90.000,C 0.000} C_DIS
LIN {X 28.344,Y -47.099,Z -108.218,A -90.000,B 90.000,C 0.000} C_DIS
LIN {X 28.047,Y -47.109,Z -108.064,A -90.000,B 90.000,C 0.000} C_DIS
LIN {X 27.716,Y -47.120,Z -107.908,A -90.000,B 90.000,C 0.000} C_DIS
LIN {X 27.238,Y -47.134,Z -107.695,A -90.000,B 90.000,C 0.000} C_DIS
LIN {X 27.084,Y -47.138,Z -107.631,A -90.000,B 90.000,C 0.000} C_DIS
LIN {X 26.914,Y -47.142,Z -107.565,A -90.000,B 90.000,C 0.000} C_DIS
LIN {X 26.595,Y -47.150,Z -107.449,A -90.000,B 90.000,C 0.000} C_DIS
LIN {X 26.273,Y -47.157,Z -107.345,A -90.000,B 90.000,C 0.000} C_DIS
LIN {X 26.144,Y -47.155,Z -107.304,A -90.000,B 90.000,C 0.000} C_DIS
LIN {X 25.774,Y -47.149,Z -107.198,A -90.000,B 90.000,C 0.000} C_DIS
LIN {X 25.614,Y -47.146,Z -107.155,A -90.000,B 90.000,C 0.000} C_DIS
LIN {X 25.335,Y -47.144,Z -107.085,A -90.000,B 90.000,C 0.000} C_DIS
LIN {X 25.047,Y -47.142,Z -107.022,A -90.000,B 90.000,C 0.000} C_DIS
LIN {X 24.176,Y -47.133,Z -106.846,A -90.000,B 90.000,C 0.000} C_DIS
LIN {X 22.848,Y -47.117,Z -106.612,A -90.000,B 90.000,C 0.000} C_DIS
LIN {X 21.954,Y -47.089,Z -106.454,A -90.000,B 90.000,C 0.000} C_DIS
LIN {X 20.891,Y -47.060,Z -106.268,A -90.000,B 90.000,C 0.000} C_DIS
LIN {X 20.407,Y -47.046,Z -106.197,A -90.000,B 90.000,C 0.000} C_DIS
LIN {X 19.973,Y -47.032,Z -106.148,A -90.000,B 90.000,C 0.000} C_DIS
LIN {X 19.433,Y -47.014,Z -106.104,A -90.000,B 90.000,C 0.000} C_DIS
LIN {X 19.207,Y -47.005,Z -106.093,A -90.000,B 90.000,C 0.000} C_DIS
LIN {X 18.962,Y -46.994,Z -106.085,A -90.000,B 90.000,C 0.000} C_DIS
LIN {X 18.320,Y -46.965,Z -106.085,A -90.000,B 90.000,C 0.000} C_DIS
LIN {X 17.968,Y -46.948,Z -106.094,A -90.000,B 90.000,C 0.000} C_DIS
LIN {X 17.610,Y -46.931,Z -106.111,A -90.000,B 90.000,C 0.000} C_DIS
LIN {X 17.151,Y -46.908,Z -106.149,A -90.000,B 90.000,C 0.000} C_DIS
LIN {X 15.519,Y -46.822,Z -106.323,A -90.000,B 90.000,C 0.000} C_DIS
LIN {X 14.831,Y -46.789,Z -106.397,A -90.000,B 90.000,C 0.000} C_DIS
LIN {X 12.609,Y -46.692,Z -106.633,A -90.000,B 90.000,C 0.000} C_DIS
LIN {X 12.334,Y -46.680,Z -106.671,A -90.000,B 90.000,C 0.000} C_DIS
LIN {X 11.783,Y -46.653,Z -106.767,A -90.000,B 90.000,C 0.000} C_DIS
LIN {X 11.477,Y -46.638,Z -106.831,A -90.000,B 90.000,C 0.000} C_DIS
LIN {X 11.289,Y -46.629,Z -106.873,A -90.000,B 90.000,C 0.000} C_DIS
LIN {X 10.780,Y -46.608,Z -107.001,A -90.000,B 90.000,C 0.000} C_DIS
LIN {X 10.350,Y -46.588,Z -107.126,A -90.000,B 90.000,C 0.000} C_DIS
LIN {X 10.173,Y -46.578,Z -107.181,A -90.000,B 90.000,C 0.000} C_DIS
LIN {X 9.300,Y -46.526,Z -107.451,A -90.000,B 90.000,C 0.000} C_DIS
LIN {X 6.380,Y -46.423,Z -108.361,A -90.000,B 90.000,C 0.000} C_DIS
LIN {X 5.389,Y -46.373,Z -108.670,A -90.000,B 90.000,C 0.000} C_DIS
LIN {X 5.197,Y -46.363,Z -108.736,A -90.000,B 90.000,C 0.000} C_DIS
LIN {X 4.912,Y -46.348,Z -108.838,A -90.000,B 90.000,C 0.000} C_DIS
LIN {X 4.423,Y -46.322,Z -109.032,A -90.000,B 90.000,C 0.000} C_DIS
LIN {X 4.116,Y -46.305,Z -109.163,A -90.000,B 90.000,C 0.000} C_DIS
LIN {X 3.755,Y -46.284,Z -109.331,A -90.000,B 90.000,C 0.000} C_DIS
LIN {X 3.484,Y -46.269,Z -109.466,A -90.000,B 90.000,C 0.000} C_DIS
LIN {X 0.747,Y -46.109,Z -110.867,A -90.000,B 90.000,C 0.000} C_DIS
LIN {X 0.225,Y -46.068,Z -111.135,A -90.000,B 90.000,C 0.000} C_DIS
LIN {X -0.051,Y -46.044,Z -111.282,A -90.000,B 90.000,C 0.000} C_DIS
LIN {X -0.329,Y -46.019,Z -111.439,A -90.000,B 90.000,C 0.000} C_DIS
LIN {X -0.697,Y -45.987,Z -111.658,A -90.000,B 90.000,C 0.000} C_DIS
LIN {X -1.111,Y -45.951,Z -111.923,A -90.000,B 90.000,C 0.000} C_DIS
LIN {X -1.621,Y -45.907,Z -112.277,A -90.000,B 90.000,C 0.000} C_DIS
LIN {X -3.396,Y -45.754,Z -113.518,A -90.000,B 90.000,C 0.000} C_DIS
LIN {X -3.521,Y -45.740,Z -113.607,A -90.000,B 90.000,C 0.000} C_DIS
LIN {X -4.039,Y -45.678,Z -113.992,A -90.000,B 90.000,C 0.000} C_DIS
LIN {X -4.256,Y -45.653,Z -114.161,A -90.000,B 90.000,C 0.000} C_DIS
LIN {X -4.612,Y -45.610,Z -114.454,A -90.000,B 90.000,C 0.000} C_DIS
LIN {X -4.844,Y -45.583,Z -114.657,A -90.000,B 90.000,C 0.000} C_DIS
LIN {X -5.599,Y -45.493,Z -115.362,A -90.000,B 90.000,C 0.000} C_DIS
LIN {X -5.743,Y -45.480,Z -115.496,A -90.000,B 90.000,C 0.000} C_DIS
LIN {X -6.113,Y -45.448,Z -115.856,A -90.000,B 90.000,C 0.000} C_DIS
LIN {X -6.227,Y -45.436,Z -115.968,A -90.000,B 90.000,C 0.000} C_DIS
LIN {X -7.175,Y -45.308,Z -116.899,A -90.000,B 90.000,C 0.000} C_DIS
LIN {X -7.175,Y -60.000,Z -116.899,A -90.000,B 90.000,C 0.000} C_DIS
LIN {X 39.370,Y -60.000,Z -122.046,A -90.000,B 90.000,C 0.000} C_DIS
LIN {X 39.370,Y -45.308,Z -122.046,A -90.000,B 90.000,C 0.000} C_DIS
LIN {X 39.371,Y -45.322,Z -121.964,A -90.000,B 90.000,C 0.000} C_DIS
LIN {X 39.359,Y -45.421,Z -121.404,A -90.000,B 90.000,C 0.000} C_DIS
LIN {X 39.350,Y -45.458,Z -121.206,A -90.000,B 90.000,C 0.000} C_DIS
LIN {X 39.317,Y -45.538,Z -120.762,A -90.000,B 90.000,C 0.000} C_DIS
LIN {X 39.285,Y -45.594,Z -120.465,A -90.000,B 90.000,C 0.000} C_DIS
LIN {X 39.268,Y -45.614,Z -120.319,A -90.000,B 90.000,C 0.000} C_DIS
LIN {X 39.184,Y -45.693,Z -119.765,A -90.000,B 90.000,C 0.000} C_DIS
LIN {X 39.024,Y -45.828,Z -118.770,A -90.000,B 90.000,C 0.000} C_DIS
LIN {X 38.953,Y -45.884,Z -118.360,A -90.000,B 90.000,C 0.000} C_DIS
LIN {X 38.871,Y -45.933,Z -117.981,A -90.000,B 90.000,C 0.000} C_DIS
LIN {X 38.805,Y -45.972,Z -117.690,A -90.000,B 90.000,C 0.000} C_DIS
LIN {X 38.709,Y -46.024,Z -117.307,A -90.000,B 90.000,C 0.000} C_DIS
LIN {X 38.642,Y -46.058,Z -117.072,A -90.000,B 90.000,C 0.000} C_DIS
LIN {X 38.527,Y -46.115,Z -116.689,A -90.000,B 90.000,C 0.000} C_DIS
LIN {X 38.463,Y -46.144,Z -116.499,A -90.000,B 90.000,C 0.000} C_DIS
LIN {X 38.393,Y -46.171,Z -116.295,A -90.000,B 90.000,C 0.000} C_DIS
LIN {X 38.309,Y -46.202,Z -116.058,A -90.000,B 90.000,C 0.000} C_DIS
LIN {X 38.253,Y -46.221,Z -115.913,A -90.000,B 90.000,C 0.000} C_DIS
LIN {X 38.099,Y -46.252,Z -115.533,A -90.000,B 90.000,C 0.000} C_DIS
LIN {X 37.914,Y -46.288,Z -115.117,A -90.000,B 90.000,C 0.000} C_DIS
LIN {X 37.858,Y -46.298,Z -115.003,A -90.000,B 90.000,C 0.000} C_DIS
LIN {X 37.773,Y -46.317,Z -114.832,A -90.000,B 90.000,C 0.000} C_DIS
LIN {X 37.702,Y -46.334,Z -114.689,A -90.000,B 90.000,C 0.000} C_DIS
LIN {X 37.540,Y -46.370,Z -114.374,A -90.000,B 90.000,C 0.000} C_DIS
LIN {X 37.287,Y -46.426,Z -113.925,A -90.000,B 90.000,C 0.000} C_DIS
LIN {X 37.019,Y -46.479,Z -113.489,A -90.000,B 90.000,C 0.000} C_DIS
LIN {X 36.806,Y -46.514,Z -113.167,A -90.000,B 90.000,C 0.000} C_DIS
LIN {X 36.608,Y -46.547,Z -112.887,A -90.000,B 90.000,C 0.000} C_DIS
LIN {X 36.569,Y -46.555,Z -112.831,A -90.000,B 90.000,C 0.000} C_DIS
LIN {X 36.353,Y -46.601,Z -112.545,A -90.000,B 90.000,C 0.000} C_DIS
LIN {X 36.268,Y -46.611,Z -112.433,A -90.000,B 90.000,C 0.000} C_DIS
LIN {X 35.937,Y -46.643,Z -112.025,A -90.000,B 90.000,C 0.000} C_DIS
LIN {X 35.034,Y -46.720,Z -110.991,A -90.000,B 90.000,C 0.000} C_DIS
LIN {X 34.781,Y -46.754,Z -110.712,A -90.000,B 90.000,C 0.000} C_DIS
LIN {X 34.630,Y -46.774,Z -110.553,A -90.000,B 90.000,C 0.000} C_DIS
LIN {X 34.421,Y -46.802,Z -110.341,A -90.000,B 90.000,C 0.000} C_DIS
LIN {X 34.176,Y -46.833,Z -110.103,A -90.000,B 90.000,C 0.000} C_DIS
LIN {X 33.797,Y -46.882,Z -109.756,A -90.000,B 90.000,C 0.000} C_DIS
LIN {X 33.423,Y -46.923,Z -109.436,A -90.000,B 90.000,C 0.000} C_DIS
LIN {X 33.381,Y -46.925,Z -109.401,A -90.000,B 90.000,C 0.000} C_DIS
LIN {X 33.164,Y -46.933,Z -109.227,A -90.000,B 90.000,C 0.000} C_DIS
LIN {X 32.785,Y -46.963,Z -108.931,A -90.000,B 90.000,C 0.000} C_DIS
LIN {X 32.472,Y -46.986,Z -108.687,A -90.000,B 90.000,C 0.000} C_DIS
LIN {X 31.076,Y -47.057,Z -107.600,A -90.000,B 90.000,C 0.000} C_DIS
LIN {X 30.892,Y -47.074,Z -107.463,A -90.000,B 90.000,C 0.000} C_DIS
LIN {X 30.710,Y -47.090,Z -107.334,A -90.000,B 90.000,C 0.000} C_DIS
LIN {X 30.494,Y -47.110,Z -107.184,A -90.000,B 90.000,C 0.000} C_DIS
LIN {X 30.104,Y -47.119,Z -106.930,A -90.000,B 90.000,C 0.000} C_DIS
LIN {X 29.895,Y -47.124,Z -106.802,A -90.000,B 90.000,C 0.000} C_DIS
LIN {X 29.572,Y -47.131,Z -106.612,A -90.000,B 90.000,C 0.000} C_DIS
LIN {X 29.306,Y -47.136,Z -106.465,A -90.000,B 90.000,C 0.000} C_DIS
LIN {X 28.960,Y -47.144,Z -106.285,A -90.000,B 90.000,C 0.000} C_DIS
LIN {X 28.570,Y -47.163,Z -106.100,A -90.000,B 90.000,C 0.000} C_DIS
LIN {X 28.057,Y -47.188,Z -105.870,A -90.000,B 90.000,C 0.000} C_DIS
LIN {X 27.845,Y -47.198,Z -105.783,A -90.000,B 90.000,C 0.000} C_DIS
LIN {X 27.643,Y -47.207,Z -105.703,A -90.000,B 90.000,C 0.000} C_DIS
LIN {X 27.360,Y -47.219,Z -105.600,A -90.000,B 90.000,C 0.000} C_DIS
LIN {X 27.257,Y -47.222,Z -105.563,A -90.000,B 90.000,C 0.000} C_DIS
LIN {X 26.767,Y -47.221,Z -105.404,A -90.000,B 90.000,C 0.000} C_DIS
LIN {X 26.437,Y -47.220,Z -105.309,A -90.000,B 90.000,C 0.000} C_DIS
LIN {X 26.210,Y -47.219,Z -105.245,A -90.000,B 90.000,C 0.000} C_DIS
LIN {X 25.821,Y -47.222,Z -105.146,A -90.000,B 90.000,C 0.000} C_DIS
LIN {X 25.473,Y -47.224,Z -105.069,A -90.000,B 90.000,C 0.000} C_DIS
LIN {X 24.571,Y -47.228,Z -104.888,A -90.000,B 90.000,C 0.000} C_DIS
LIN {X 23.885,Y -47.231,Z -104.767,A -90.000,B 90.000,C 0.000} C_DIS
LIN {X 22.427,Y -47.198,Z -104.510,A -90.000,B 90.000,C 0.000} C_DIS
LIN {X 21.237,Y -47.176,Z -104.301,A -90.000,B 90.000,C 0.000} C_DIS
LIN {X 20.694,Y -47.165,Z -104.221,A -90.000,B 90.000,C 0.000} C_DIS
LIN {X 20.638,Y -47.164,Z -104.213,A -90.000,B 90.000,C 0.000} C_DIS
LIN {X 20.190,Y -47.152,Z -104.164,A -90.000,B 90.000,C 0.000} C_DIS
LIN {X 19.591,Y -47.133,Z -104.114,A -90.000,B 90.000,C 0.000} C_DIS
LIN {X 19.300,Y -47.124,Z -104.099,A -90.000,B 90.000,C 0.000} C_DIS
LIN {X 19.020,Y -47.114,Z -104.090,A -90.000,B 90.000,C 0.000} C_DIS
LIN {X 18.325,Y -47.090,Z -104.089,A -90.000,B 90.000,C 0.000} C_DIS
LIN {X 17.915,Y -47.076,Z -104.098,A -90.000,B 90.000,C 0.000} C_DIS
LIN {X 17.508,Y -47.061,Z -104.118,A -90.000,B 90.000,C 0.000} C_DIS
LIN {X 16.979,Y -47.040,Z -104.161,A -90.000,B 90.000,C 0.000} C_DIS
LIN {X 15.989,Y -47.006,Z -104.267,A -90.000,B 90.000,C 0.000} C_DIS
LIN {X 14.614,Y -46.944,Z -104.415,A -90.000,B 90.000,C 0.000} C_DIS
LIN {X 13.129,Y -46.873,Z -104.572,A -90.000,B 90.000,C 0.000} C_DIS
LIN {X 12.391,Y -46.847,Z -104.651,A -90.000,B 90.000,C 0.000} C_DIS
LIN {X 12.054,Y -46.834,Z -104.697,A -90.000,B 90.000,C 0.000} C_DIS
LIN {X 11.433,Y -46.808,Z -104.804,A -90.000,B 90.000,C 0.000} C_DIS
LIN {X 11.104,Y -46.794,Z -104.872,A -90.000,B 90.000,C 0.000} C_DIS
LIN {X 10.848,Y -46.781,Z -104.928,A -90.000,B 90.000,C 0.000} C_DIS
LIN {X 10.285,Y -46.752,Z -105.069,A -90.000,B 90.000,C 0.000} C_DIS
LIN {X 9.788,Y -46.724,Z -105.212,A -90.000,B 90.000,C 0.000} C_DIS
LIN {X 9.581,Y -46.712,Z -105.275,A -90.000,B 90.000,C 0.000} C_DIS
LIN {X 9.214,Y -46.693,Z -105.389,A -90.000,B 90.000,C 0.000} C_DIS
LIN {X 6.452,Y -46.532,Z -106.246,A -90.000,B 90.000,C 0.000} C_DIS
